tonAirBeforeStart2(IN:=eRunningStateFeeder=E_WickFeederSorterState.eSorting, PT:=T#2S);
tonAirAfterStop(IN:=eRunningStateFeeder=E_WickFeederSorterState.eSleeveFull, PT:=T#2S);

tonbSeparatorPos1AndNotbWickAtSleve1(IN:=bSeparatorPos1 AND NOT bWickAtSleve1,PT:=T#3S);
tonbSeparatorPos2AndNotbWickAtSleve2(IN:=bSeparatorPos2 AND NOT bWickAtSleve2,PT:=T#3S);
tonbSeparatorPos1(IN:=bSeparatorPos1,PT:=T#300MS);
tonbSeparatorPos2(IN:=bSeparatorPos2,PT:=T#300MS);

tobbSleve1SeparatorIn(IN:=bSleve1SeparatorIn,PT:=T#1S);
tobbSleve2SeparatorIn(IN:=bSleve2SeparatorIn,PT:=T#1S);
fbbQueFullAtSleve1 (bIN:=	bQueFullAtSleve1,	tFilterTimeOn:=T#300MS, tFilterTimeOff:=T#300MS, 	bOUT=> );										
fbbQueFullAtSleve2 (bIN:=	bQueFullAtSleve2,	tFilterTimeOn:=T#300MS, tFilterTimeOff:=T#300MS, 	bOUT=> );										
fbbWickAtPipe 		(bIN:=	bWickAtPipe,		tFilterTimeOn:=T#100MS, tFilterTimeOff:=T#30MS,		bOUT=> );	
fbbNotWickAtPipe 	(bIN:=	NOT bWickAtPipe AND iSortingCase=35,		tFilterTimeOn:=T#2S, tFilterTimeOff:=T#100MS,		bOUT=> );	
									
tonCaseA			(IN:=iSortingCase = 20 , PT:=T#600MS);
tonCaseB			(IN:=iSortingCase = 35 , PT:=T#300MS);
tonCaseC			(IN:=iSortingCase = 20 , PT:=T#600MS);
tonCaseD			(IN:=iSortingCase = 20 , PT:=T#600MS);
//prszesunęcie wartosci czujnika po buforu opoznenia 

TimerOn (IN := NOT bImpOn, PT := T#10MS);
IF TimerOn.Q THEN
	bImpOn := TRUE;
END_IF
TimerOff (IN := bImpOn, PT := T#10MS);
IF TimerOff.Q THEN
	bImpON := FALSE;
END_IF

tonHammer1Down(IN:= bHammer1Down, PT:=T#200MS);
tonHammer2Down(IN:= bHammer2Down, PT:=T#200MS);

(** Dodatkowy timer przy zatrzymywaniu**)
tonStoppingTime( IN:= eState= E_Station.eStopping, PT:=T#2S);
END_ACTION

ACTION ACT_Warning:
 //Warning czujnik poziomu	
 	tonLowLevelSensor( IN:=( NOT  bWheelLevelSensor (*OR NOT bQueFullAfterWheelSensor*) OR NOT bQueFullSensor) AND bRun, PT:= T#5S);
 	
 	IF tonLowLevelSensor.Q THEN
 		bWarning				:= TRUE;
	ELSE
		bWarning				:= FALSE;
 	END_IF
END_ACTION

END_FUNCTION_BLOCK

// ---- POUs/P08_CapSorter.TcPOU
(*
Nazwa:			P08_CapFeeder
Opis:			Stacja podajnika nasadek
Wersja:			v0.2
Data:			2024-01-12
Autor:			DP
Urzadzenia:		
Konfiguracja:	
Info:

*)
PROGRAM P08_CapSorter
VAR_INPUT
	IbCapSorterGateScrewerSensor 			:BOOL;			
	IbCapSorterGateWeightSensor				:BOOL;
	//WEJSCIA I WYJSCIA SPRZETOWE
	IbCapSorterDragHomingSensor 			 :BOOL;						// Czujnik bazowania
	QbCapSorterDragActuator               	 :BOOL;						// Siłownikiem przeciągania 
	IbCapSorterDragUpSensor 				 :BOOL;						// Czujnik
	IbCapSorterDragDownSensor 				 :BOOL;						// Czujnik
	                                         
	QbCapSorterDragLeadBefore1Actuator       :BOOL;						// Siłownikiem prowadzenia przed 
	IbCapSorterDragLeadBefore1UpSensor 	 	 :BOOL;						// Czujnik
 	IbCapSorterDragLeadBefore2UpSensor 	 	 :BOOL;						// Czujnik			
	QbCapSorterDragLeadAfter1Actuator        :BOOL;						// Siłownikiem prowadzenia za
	IbCapSorterDragLeadAfter1UpSensor 	 	 :BOOL;						// Czujnik
 	IbCapSorterDragLeadAfter2UpSensor 	 	 :BOOL;						// Czujnik			

END_VAR
VAR
	
	(*******PRZECIAGANIE**********)
	eCapSorterDragStation						: E_Station;
	eCapSorterDragRunningStation				: E_DragStationState;
	fbCapSorterDragState						: FB_State;
	fbCapSorterDragStation						: FB_FormsDragStepper;	
	
	

	
	
	//Pomocnicze
	tofCapSorterDragEnable					: TOF;
	
	//Stoper
	QbCapSorterStoperActuator				: BOOL;				// bit to wysterowania sygnału stopera	
	tpStoperTimerOn							: TP;				// timer do generowania impulsu
	fbStoperSensorDelay						: FB_InputFilter;	// filtr do generowania sygnału 
	lrCapSorterStoperPosition						: LREAL;	
	rtCapSorterStoperDraging: R_TRIG;
	rtCapSorterStoperEndingOfDraging: R_TRIG;	
	//Inne
	bTemp: BOOL;

	rtCapSorterStoperPackMLStarting: R_TRIG;
	bCapSorterStoperWaitingForSensor: BOOL;
	bCapSorterStoperActuatorDelay: BOOL;
	tonbCapSorterStoperActuatorDelay: TON;
	
	//ManualStoper
	rtManualMode	: R_TRIG;
	ftManualMode	: F_TRIG;	
	bCapSorterStoperActuatorLastState	:BOOL;
	
END_VAR

//bCapSorterDisable:=VIS.bCapPuttedCheckIgnoreErrors;


tofCapSorterDragEnable(IN:= GVL.bCapSorterDragEnable, PT:= T#5S);
aLimits();
aStoper();
aDragStation();
aCapSorterWarnings();


(********* GENEROWANIE STANU STACJI DO WIZKI**********)
fbCapSorterDragState(
	eState:=eCapSorterDragStation, 
	bRun:=VIS.bCapSorterDragRun,
	eFormsDragingRunningState:=eCapSorterDragRunningStation, 
	sStateDesc=> VIS.sCapSorterDragState,
	iState=>VIS.iCapSorterDragState);
(***** KONIEC GENEROWANIE STANU STACJI DO WIZKI*******)



IF fbCapSorterDragStation.bCycleDone AND bManualMode THEN
	VIS.bCapSorterDragRun 						:= FALSE;
	GVL.bCapSorterDragPrepareRun				:= FALSE;
END_IF

ACTION aCapSorterWarnings:

//Warning 0
IF stCapSorterRead.eReservedSignals.iReserved20.0 AND NOT CapSorterWarning[0].bWarning THEN
	CapSorterWarning[0].bWarning										:=TRUE;
	CapSorterWarning[0].udiWarningCode									:=41;
	CapSorterWarning[0].sDescription									:='Sorter nasadek | Brak nasadek w zasobniku';
ELSIF NOT stCapSorterRead.eReservedSignals.iReserved20.0 THEN//AND CapSorterWarning[0].bAcknowledge THEN
	CapSorterWarning[0].bWarning										:=FALSE;
	CapSorterWarning[0].bAcknowledge									:=FALSE;
	VIS.uliWarningAcknowledge.27										:=FALSE;
ELSIF CapSorterWarning[0].bAcknowledge THEN                               
	CapSorterWarning[0].bAcknowledge									:=TRUE;
END_IF

//Warning 1
IF stCapSorterRead.eReservedSignals.iReserved20.1 AND NOT CapSorterWarning[1].bWarning THEN
	CapSorterWarning[1].bWarning										:=TRUE;
	CapSorterWarning[1].udiWarningCode									:=42;
	CapSorterWarning[1].sDescription									:='Sorter nasadek | Brak nasadek na stole - sprawdź transporter pośredni';
ELSIF NOT stCapSorterRead.eReservedSignals.iReserved20.1 AND CapSorterWarning[1].bAcknowledge THEN
	CapSorterWarning[1].bWarning										:=FALSE;
	CapSorterWarning[1].bAcknowledge									:=FALSE;
	VIS.uliWarningAcknowledge.28										:=FALSE;
ELSIF CapSorterWarning[1].bAcknowledge THEN
	CapSorterWarning[1].bAcknowledge									:=TRUE;
END_IF

//Warning 2
IF stCapSorterRead.eReservedSignals.iReserved20.2 AND NOT CapSorterWarning[2].bWarning THEN
	CapSorterWarning[2].bWarning										:=TRUE;
	CapSorterWarning[2].udiWarningCode									:=43;
	CapSorterWarning[2].sDescription									:='Sorter nasadek | Niepobrana nasadka przez chwytak 1';
ELSIF NOT stCapSorterRead.eReservedSignals.iReserved20.1 AND CapSorterWarning[2].bAcknowledge THEN
	CapSorterWarning[2].bWarning										:=FALSE;
	CapSorterWarning[2].bAcknowledge									:=FALSE;
	VIS.uliWarningAcknowledge.29										:=FALSE;
ELSIF CapSorterWarning[2].bAcknowledge THEN
	CapSorterWarning[2].bAcknowledge									:=TRUE;
END_IF

//Warning 3
IF stCapSorterRead.eReservedSignals.iReserved20.3 AND NOT CapSorterWarning[3].bWarning THEN
	CapSorterWarning[3].bWarning										:=TRUE;
	CapSorterWarning[3].udiWarningCode									:=44;
	CapSorterWarning[3].sDescription									:='Sorter nasadek | Niepobrana nasadka przez chwytak 2';
ELSIF NOT stCapSorterRead.eReservedSignals.iReserved20.1 AND CapSorterWarning[3].bAcknowledge THEN
	CapSorterWarning[3].bWarning										:=FALSE;
	CapSorterWarning[3].bAcknowledge									:=FALSE;
	VIS.uliWarningAcknowledge.30										:=FALSE;
ELSIF CapSorterWarning[3].bAcknowledge THEN
	CapSorterWarning[3].bAcknowledge									:=TRUE;
END_IF

//Warning 4
IF stCapSorterRead.eReservedSignals.iReserved20.4 AND NOT CapSorterWarning[4].bWarning THEN
	CapSorterWarning[4].bWarning										:=TRUE;
	CapSorterWarning[4].udiWarningCode									:=45;
	CapSorterWarning[4].sDescription									:='Sorter nasadek | Niepobrana nasadka przez chwytak 3';
ELSIF NOT stCapSorterRead.eReservedSignals.iReserved20.1 AND CapSorterWarning[4].bAcknowledge THEN
	CapSorterWarning[4].bWarning										:=FALSE;
	CapSorterWarning[4].bAcknowledge									:=FALSE;
	VIS.uliWarningAcknowledge.31										:=FALSE;
ELSIF CapSorterWarning[4].bAcknowledge THEN
	CapSorterWarning[4].bAcknowledge									:=TRUE;
END_IF

//Warning 5
IF stCapSorterRead.eReservedSignals.iReserved20.5 AND NOT CapSorterWarning[5].bWarning THEN
	CapSorterWarning[5].bWarning										:=TRUE;
	CapSorterWarning[5].udiWarningCode									:=46;
	CapSorterWarning[5].sDescription									:='Sorter nasadek | Niepobrana nasadka przez chwytak 4';	
ELSIF NOT stCapSorterRead.eReservedSignals.iReserved20.1 AND CapSorterWarning[5].bAcknowledge THEN
	CapSorterWarning[5].bWarning										:=FALSE;
	CapSorterWarning[5].bAcknowledge									:=FALSE;
	VIS.uliWarningAcknowledge.32										:=FALSE;
ELSIF CapSorterWarning[5].bAcknowledge THEN
	CapSorterWarning[5].bAcknowledge									:=TRUE;
END_IF
END_ACTION

ACTION aDragStation:
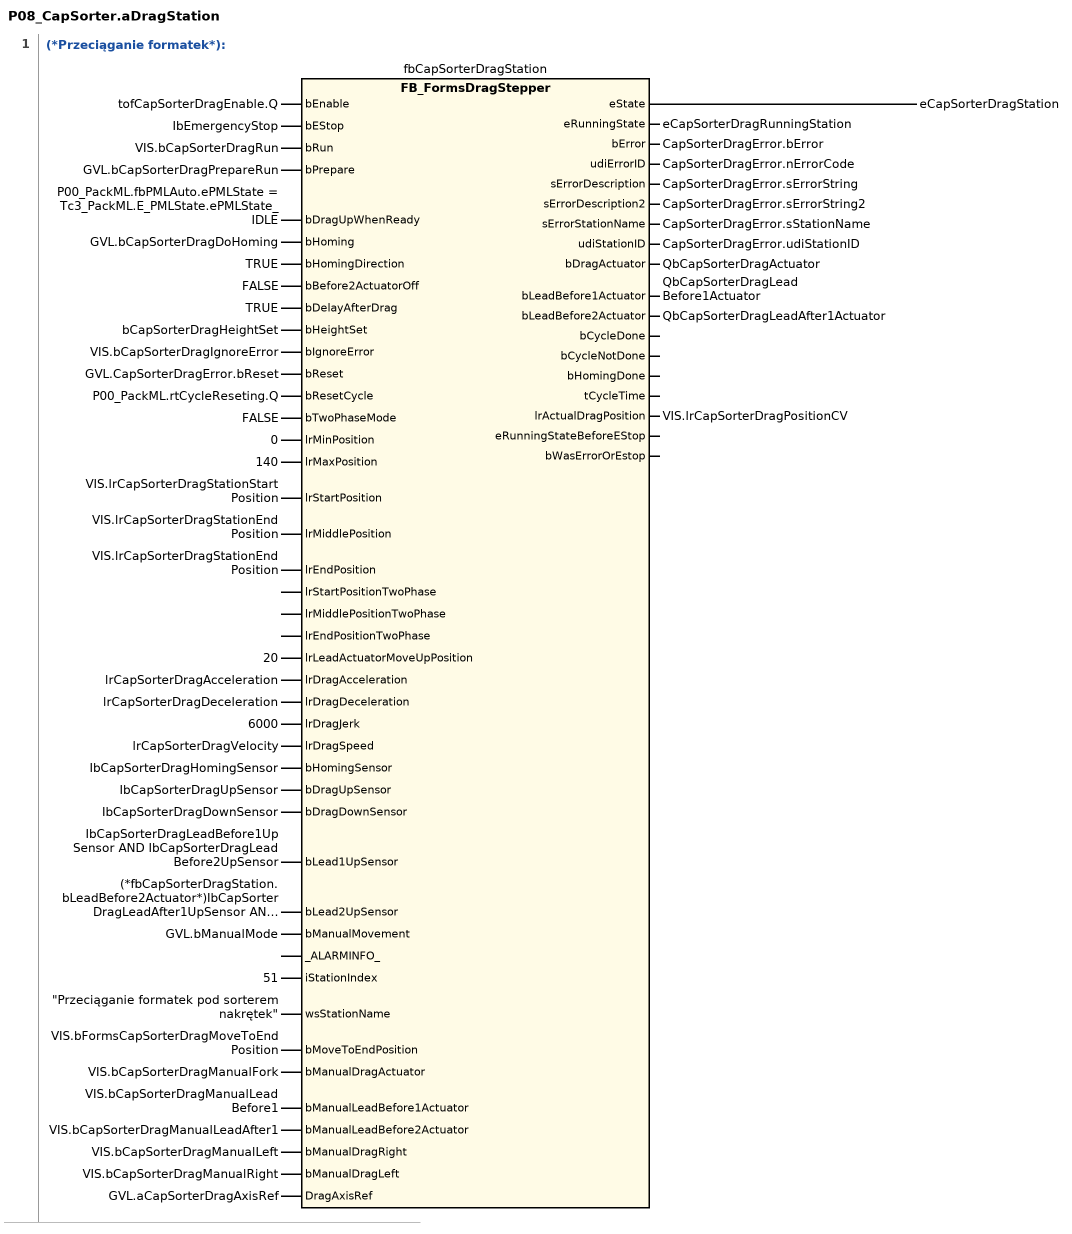
// NETWORK 1
// label: (*Przeciąganie formatek*)
fbCapSorterDragStation(
    bEnable := tofCapSorterDragEnable.Q,
    bEStop := IbEmergencyStop,
    bRun := VIS.bCapSorterDragRun,
    bPrepare := GVL.bCapSorterDragPrepareRun,
    bDragUpWhenReady := P00_PackML.fbPMLAuto.ePMLState = Tc3_PackML.E_PMLState.ePMLState_IDLE,
    bHoming := GVL.bCapSorterDragDoHoming,
    bHomingDirection := TRUE,
    bBefore2ActuatorOff := FALSE,
    bDelayAfterDrag := TRUE,
    bHeightSet := bCapSorterDragHeightSet,
    bIgnoreError := VIS.bCapSorterDragIgnoreError,
    bReset := GVL.CapSorterDragError.bReset,
    bResetCycle := P00_PackML.rtCycleReseting.Q,
    bTwoPhaseMode := FALSE,
    lrMinPosition := 0,
    lrMaxPosition := 140,
    lrStartPosition := VIS.lrCapSorterDragStationStartPosition,
    lrMiddlePosition := VIS.lrCapSorterDragStationEndPosition,
    lrEndPosition := VIS.lrCapSorterDragStationEndPosition,
    lrLeadActuatorMoveUpPosition := 20,
    lrDragAcceleration := lrCapSorterDragAcceleration,
    lrDragDeceleration := lrCapSorterDragDeceleration,
    lrDragJerk := 6000,
    lrDragSpeed := lrCapSorterDragVelocity,
    bHomingSensor := IbCapSorterDragHomingSensor,
    bDragUpSensor := IbCapSorterDragUpSensor,
    bDragDownSensor := IbCapSorterDragDownSensor,
    bLead1UpSensor := IbCapSorterDragLeadBefore1UpSensor AND IbCapSorterDragLeadBefore2UpSensor,
    bLead2UpSensor := (*fbCapSorterDragStation.bLeadBefore2Actuator*)IbCapSorterDragLeadAfter1UpSensor AND IbCapSorterDragLeadAfter2UpSensor,
    bManualMovement := GVL.bManualMode,
    iStationIndex := 51,
    wsStationName := "Przeciąganie formatek pod sorterem nakrętek",
    bMoveToEndPosition := VIS.bFormsCapSorterDragMoveToEndPosition,
    bManualDragActuator := VIS.bCapSorterDragManualFork,
    bManualLeadBefore1Actuator := VIS.bCapSorterDragManualLeadBefore1,
    bManualLeadBefore2Actuator := VIS.bCapSorterDragManualLeadAfter1,
    bManualDragRight := VIS.bCapSorterDragManualLeft,
    bManualDragLeft := VIS.bCapSorterDragManualRight,
    DragAxisRef := GVL.aCapSorterDragAxisRef,
    eRunningState => eCapSorterDragRunningStation,
    bError => CapSorterDragError.bError,
    udiErrorID => CapSorterDragError.nErrorCode,
    sErrorDescription => CapSorterDragError.sErrorString,
    sErrorDescription2 => CapSorterDragError.sErrorString2,
    sErrorStationName => CapSorterDragError.sStationName,
    udiStationID => CapSorterDragError.udiStationID,
    bDragActuator => QbCapSorterDragActuator,
    bLeadBefore1Actuator => QbCapSorterDragLeadBefore1Actuator,
    bLeadBefore2Actuator => QbCapSorterDragLeadAfter1Actuator,
    lrActualDragPosition => VIS.lrCapSorterDragPositionCV); // FB_FormsDragStepper
eCapSorterDragStation := fbCapSorterDragStation.eState;
END_ACTION

ACTION aLimits:
//
IF 	VIS.lrCapSorterDragStationStartPosition		= 0		THEN	VIS.lrCapSorterDragStationStartPosition	:=	7;		END_IF;
IF 	VIS.lrCapSorterDragStationEndPosition		= 0		THEN	VIS.lrCapSorterDragStationEndPosition		:=	142;	END_IF;
END_ACTION

ACTION aStoper:
(*
Nazwa:			aStoper
Opis:			Stoper spowalniania formatek
Wersja:			v0.1
Data:			2024-03-21
Autor:			DP
Urzadzenia:		
Konfiguracja:	
Info:

*)


// 0 - Przliczanie od predkości przeciagania				   
lrCapSorterStoperPosition	 :=	(188.25 * EXPT(lrCapSorterDragVelocity,-0.404));
	

// 1 - Wysuwanie stopera na koniec przesuwania gdy pracuje
rtCapSorterStoperDraging(CLK:=  
								P08_CapSorter.fbCapSorterDragStation.eRunningState = E_DragStationState.eDraging AND 
								((P00_PackML.fbPMLAuto.ePMLState = E_PMLState.ePMLState_STOPPING) OR  (P00_PackML.fbPMLAuto.ePMLState = E_PMLState.ePMLState_EXECUTE)) AND
						   		P08_CapSorter.fbCapSorterDragStation.lrActualDragPosition > lrCapSorterStoperPosition+20 
						,Q=>);
						
IF rtCapSorterStoperDraging.Q THEN
	QbCapSorterStoperActuator	:= TRUE;
END_IF


									
// 2 - Sygnał czekania na czujnik formatek
rtCapSorterStoperPackMLStarting (CLK:=  	
											(P00_PackML.fbPMLAuto.ePMLState = E_PMLState.ePMLState_STARTING)
								,Q=>);

								

//rtCapSorterStoperEndingOfDraging(CLK:=  	P08_CapSorter.fbCapSorterDragStation.eRunningState = E_DragStationState.eDraged AND 
rtCapSorterStoperEndingOfDraging(CLK:=  	P08_CapSorter.fbCapSorterDragStation.eRunningState = E_DragStationState.eDragingDone AND 
											((P00_PackML.fbPMLAuto.ePMLState = E_PMLState.ePMLState_STOPPING) OR  (P00_PackML.fbPMLAuto.ePMLState = E_PMLState.ePMLState_EXECUTE))
								,Q=>);
						

IF rtCapSorterStoperEndingOfDraging.Q OR rtCapSorterStoperPackMLStarting.Q THEN
	bCapSorterStoperWaitingForSensor	:=	TRUE;	
END_IF							

// 3 - Wyłączanie stopera
IF NOT bDosingTwoPhases THEN
	IF bCapSorterStoperWaitingForSensor AND P00_PackML.fbIbCapSorterFourthFormCheckFormSensor.bOut THEN	
		bCapSorterStoperActuatorDelay	:=	TRUE;
	END_IF
ELSE
	IF bCapSorterStoperWaitingForSensor (*AND MAIN.IbCapSorterFourthFormCheckFormSensor*) AND iCapSorterDragFormCounter >=1 AND P00_ReadRFIDCard.bReadedCardCapSorter THEN	
		bCapSorterStoperActuatorDelay	:=	TRUE;
	END_IF
END_IF

IF 	nFormTransportersBeforeScrewerVelocitySV < 610 AND NOT bDosingTwoPhases THEN
	tonbCapSorterStoperActuatorDelay(IN:=bCapSorterStoperActuatorDelay, PT:=T#1S150MS);
ELSE
	tonbCapSorterStoperActuatorDelay(IN:=bCapSorterStoperActuatorDelay, PT:=T#790MS);//990
END_IF

IF tonbCapSorterStoperActuatorDelay.Q THEN
	bCapSorterStoperActuatorDelay		:=	FALSE;
	bCapSorterStoperWaitingForSensor	:=	FALSE;
	QbCapSorterStoperActuator			:=	FALSE;
END_IF


//Manual
rtManualMode	(CLK:=bManualMode,	Q=>);
ftManualMode	(CLK:=bManualMode,	Q=>);
IF rtManualMode.Q THEN
	bCapSorterStoperActuatorLastState	:=	QbCapSorterStoperActuator;
	VIS.bCapSorterStoperManualActuator	:=	QbCapSorterStoperActuator;
END_IF
IF bManualMode THEN
	QbCapSorterStoperActuator			:=	VIS.bCapSorterStoperManualActuator;
END_IF
IF ftManualMode.Q THEN
	QbCapSorterStoperActuator			:= bCapSorterStoperActuatorLastState;
END_IF
// Koniec Manual
END_ACTION

END_PROGRAM

// ---- POUs/P01_PucksInserter.TcPOU
(*
Nazwa:			P01_PucksInserter
Opis:			Stacja podajnika opakowań
Wersja:			v0.1
Data:			2025-02-04
Autor:			DP
Urzadzenia:		
Konfiguracja:	
Info:

*)
PROGRAM P01_PucksInserter
VAR_INPUT

	//52N6.1 Pneumatyka IO
	IbPucksInserterLevelSensor					:BOOL;			// Czujnik kolejki butelki
	IbPucksInserterWheelEntrySensor				:BOOL;			// Czujnik   pierwszego slotu w karuzeli (to 
	IbPucksInserterWheelExitSensor				:BOOL;			// Czujnik
	IbPucksInserterFormGateBeforeSensor 		:BOOL;			// Czujnik przed szlabanem formatek
	IbPucksInserterFormGateAfterSensor 			:BOOL;			// Czujnik za szlabanem formatek	
 	IbPucksInserterHammerUpSensor				:BOOL;			// Czujnik położenia siłownika - góra
	IbPucksInserterHammerDownSensor				:BOOL;			// Czujnik polożenia siłowniak - dół
	IbPucksInserterTrayOnSensor					:BOOL;			// Czujnik tacka wysunieta
	//52N6.2 Pneumatyka IO	
	IbPucksInserterTrayOffSensor				:BOOL;			// Czujnik tacka schowana
	IbPucksInserterFormPositioningOnSensor		:BOOL;			// Czujnik wysuniecia siłownika pozycjonujacego formatke
	IbPucksInserterFormPositioningOffSensor		:BOOL;			// Czujnik schowania siłownika pozycjonujacego formatke
	IbPucksInserterGate1OnSensor				:BOOL;			// Czujnik otwarcia 1 szlabanu (Lewy)
	IbPucksInserterGate1OffSensor				:BOOL;			// Czujnik zamknięcia 1 szlabanu (Lewy) 
	IbPucksInserterGate2OnSensor				:BOOL;			// Czujnik otwarcia 2 szlabanu 
	IbPucksInserterGate2OffSensor				:BOOL;			// Czujnik zamknięcia 2 szlabanu (Prawy) 
	IbPucksInserterHomingSensor					:BOOL;			// Czujnik bazowania
	
	//Inne
	IbPucksInserterNotInsertedSensor			:BOOL;			// Czujnik źle włozonej butelki za stacją	
	
	IbPucksInserterPushTablesSensor				:BOOL;
END_VAR

VAR

	//BC3 
	IbPucksInserterFuseDrivesOK					AT %I*: BOOL; 			// Zabezpieczenie serwa
	IbPucksInserterTransporter1OK				AT %I*: BOOL; 			// Bezpiecznik silnikowe napędu transportera 1
	IbPucksInserterTransporter2OK				AT %I*: BOOL; 			// Bezpiecznik silnikowe napędu transportera 2	
	IbPucksInserterFuseFB1OK					AT %I*: BOOL;			// Bezpiecznik FB1 przepalony
	QbPucksInserterHammerHeightUpCmd 			AT %Q*: BOOL; 			// Wyjście sterujące podnośnikiem
	QbPucksInserterHammerHeightDownCmd 			AT %Q*: BOOL; 			// Wyjście sterujące podnośnikiem
	//GVL_IO QbPickInserterDoorsClose			AT %Q*:BOOL;			// Rozkaz zamkniecia
	QudiPucksInserterHammerHeightEncoderSetCV	AT %Q*: UDINT;			// Enkoder - Set Counter value
	QbPucksInserterHammerHeightEncoderSetC		AT %Q*: BOOL; 			// Enkoder - Set Counter 
	IudiPucksInserterHammerHeightEncoderCV 		AT %I*: UDINT;	 		// Enkoder - Counter value
	IbPucksInserterHammerHeightEncoderSetCDone	AT %I*: BOOL; 			// Enkoder - Set Counter done

	//DI5
	//GVL_IO IbPucksInserterDoorsOpen	{warning 'PI'}	AT %I*	:BOOL;	//Otwarte drzwi podajnika opakowań
	//GLV_IO etop 0
	//GLV_IO etop 1
	//GLV_IO stop
	//GLV_IO start
	//Safety reset

	//DO4
	//Lamps green
	//Lamps blue

	fbPucksInserter						  	: FB_PucksInserter;		// Bloczek do obsługi stacji podajnika butelek
	fbTurnTable								: FB_MitsubishiInverter; 	//Bloczek do obsługi falownika stołu obrotewego
	
	ePucksInserterStationState				: E_Station;
	ePucksInserterRunningState				: E_PuckInserterState;
	fbPucksInserterState					: FB_State;
	
	ePucksInserterTurnTableState			: E_Station;
	ePucksInserterTurnTableRunningState		: E_ConveyorState;
	fbBottleSorterTurnTableState			: FB_State;
	
	fbGatePucksInserter						: FB_SpringGateV2;
	
	//Wyjścia sterujące
	QbPucksInserterHammer					:BOOL;			// Wbijak
	QbPucksInserterTray						:BOOL;			// Ruchomy blat (tacka)
	QbPucksInserterGate1					:BOOL;			// Szlaban 1 (lewy)
	QbPucksInserterGate2					:BOOL;			// Szlaban 2 (prawy)
	QbPucksInserterFormGate					:BOOL;			// Szlaban formatki
	QbPucksInserterFormPositioning			:BOOL;			// Pozycjonowanie formatki

	// Stół obrotowy
	uiPucksInserterTurnTableSW					AT %I*: UINT;
	uiPucksInserterTurnTableActualVelocity		AT %I*: UDINT;
	uiPucksInserterTurnTableCW  				AT %Q*: UINT;
	udiPucksInserterTurnTableVelocity			AT %Q*: UDINT;
	
	// Transporter
	uiPucksInserterConveyorSW					AT %I*: UINT;
	uiPucksInserterConveyorActualVelocity		AT %I*: UDINT;
	uiPucksInserterConveyorCW  					AT %Q*: UINT;
	udiPucksInserterConveyorVelocity			AT %Q*: UDINT;	
	IbPucksInserterConveyorWcState				AT %I*: BOOL;
	
	// Serwo
	// GVL axis
	diPucksInserterWheelZPhaseOffset			AT %I*: DINT; // Offset serwa Z


	// Bazowanie
	tonPucksInserterEnable	: TON;
	rtEnable	: R_TRIG;
	
	//testowe
	bTest :BOOL;
	bTest2 :BOOL;	
	bTestHomingPI:BOOL;
	bPITest:BOOL;
	 
	//Stół pchający    //Vasyl 27.05
	fbPushTable_m1: FB_MitsubishiInverter;
	fbPushTable_m2: FB_MitsubishiInverter;
	fbPushTable_m3: FB_MitsubishiInverter;	
	
	QnPucksInserterPushTable_m1_VelocitySV 						AT %Q*: UDINT; 	
	InPucksInserterPushTable_m1_VelocityCV 						AT %I*: UDINT;	
	InPucksInserterPushTable_m1_STW 							AT %I*: UINT; 	
	QnPucksInserterPushTable_m1_CTW 							AT %Q*: UINT;  	
	InPucksInserterPushTable_m1_ErrorCode 						AT %I*: UINT;	
	
	QnPucksInserterPushTable_m2_VelocitySV 						AT %Q*: UDINT; 	
	InPucksInserterPushTable_m2_VelocityCV 						AT %I*: UDINT;	
	InPucksInserterPushTable_m2_STW 							AT %I*: UINT; 
	QnPucksInserterPushTable_m2_CTW 							AT %Q*: UINT;  	
	InPucksInserterPushTable_m2_ErrorCode 						AT %I*: UINT;	
	
	QnPucksInserterPushTable_m3_VelocitySV 						AT %Q*: UDINT; 	
	InPucksInserterPushTable_m3_VelocityCV 						AT %I*: UDINT; 	
	InPucksInserterPushTable_m3_STW 							AT %I*: UINT; 
	QnPucksInserterPushTable_m3_CTW 							AT %Q*: UINT;  	
	InPucksInserterPushTable_m3_ErrorCode 						AT %I*: UINT;	

	
	fbPucksInserterPushTableState			: FB_State;
	ePucksInserterPushTableState			: E_Station;
	ePucksInserterPushTableRunningState		: E_PuckInserterState;
	
	fbPucksInserterPushTableRollerState			: FB_State;
	ePucksInserterPushTableRollerState			: E_Station;
	ePucksInserterPushTableRollerRunningState	: E_PuckInserterState;
END_VAR

aWarning();
aPucksInserter();
aTurntable(); 
aGateTime();
aGate();
aPushTable();

//VIS.nPucksInserterTurnTableVelocityCV := uiPucksInserterTurnTableActualVelocity;
VIS.nPucksInserterConveyorVelocityCV:=uiPucksInserterConveyorActualVelocity;
VIS.uiPucksInserterPushTable_m1_Velocity:=UDINT_TO_INT(InPucksInserterPushTable_m1_VelocityCV);
VIS.uiPucksInserterPushTable_m2_Velocity:=UDINT_TO_INT(InPucksInserterPushTable_m2_VelocityCV);
VIS.uiPucksInserterPushTable_m3_Velocity:=UDINT_TO_INT(InPucksInserterPushTable_m3_VelocityCV);

(* BAZOWANIE - ZMIAN*)
tonPucksInserterEnable (IN:=fbPucksInserter.bEnable,PT:=T#5S); (*Dodany ton bo Wizka zjebnie wgrywa zmienne, najpierw włacza Enabla a potem dopiero wybiera recepture*)
rtEnable(CLK:=tonPucksInserterEnable.Q,Q=>);
IF rtEnable.Q AND (P00_PackML.fbPMLAuto.ePMLState = E_PMLState.ePMLState_IDLE OR P00_PackML.fbPMLAuto.ePMLState = E_PMLState.ePMLState_EXECUTE)   THEN
	VIS.bPucksInserterHeightSet:=TRUE;
ELSIF fbPucksInserter.eState=E_Station.eHomingDone  OR VIS.bErrorOccure THEN
 	VIS.bPucksInserterHeightSet:=FALSE;
END_IF
(*KONIEC BAZOWANIE - ZMIANA*)


(********KASOWANIE ROZKAZÓW CYKLI*********)
IF fbPucksInserter.bCycleDone AND bManualMode THEN
	VIS.bPucksInserterRun := FALSE;
END_IF

(*
IF bPITest AND NOT VIS.bPucksInserterRun THEN
	VIS.bPucksInserterRun := TRUE;
END_IF
IF VIS.bPucksInserterRun AND bPITest AND fbPucksInserter.bCycleDone THEN
	VIS.bPucksInserterRun := FALSE;	
END_IF*)


fbPucksInserterState(
	eState									:= ePucksInserterStationState,
	bRun									:= VIS.bPucksInserterRun,
	eBottleSorterRunningState				:= ePucksInserterRunningState,
	sStateDesc								=> VIS.sPucksInserterState,
	iState									=> VIS.iPucksInserterState);
	
fbPucksInserterPushtableState(
	eState									:= ePucksInserterPushTableState,
    bRun						            := gvl.bPucksInserterPushTable_m1_Run OR vis.bPucksInserterPushTable_m1_ManualCmdStart,
    eBottleSorterRunningState	            := ePucksInserterPushTableRunningState,
    sStateDesc					            => VIS.sPucksInserterPushTableState,
    iState						            => VIS.iPucksInserterPushTableState);
	
fbPucksInserterPushTableRollerState(
	eState									:= ePucksInserterPushTableRollerState,	
    bRun						            := gvl.bPucksInserterPushTable_m2_Run OR vis.bPucksInserterPushTable_m2_ManualCmdStart,	
    eBottleSorterRunningState	            := ePucksInserterPushTableRollerRunningState,	
    sStateDesc					            => VIS.sPucksInserterPushTableRollerState,	
    iState						            => VIS.iPucksInserterPushTableRollerState);

ACTION aGate:
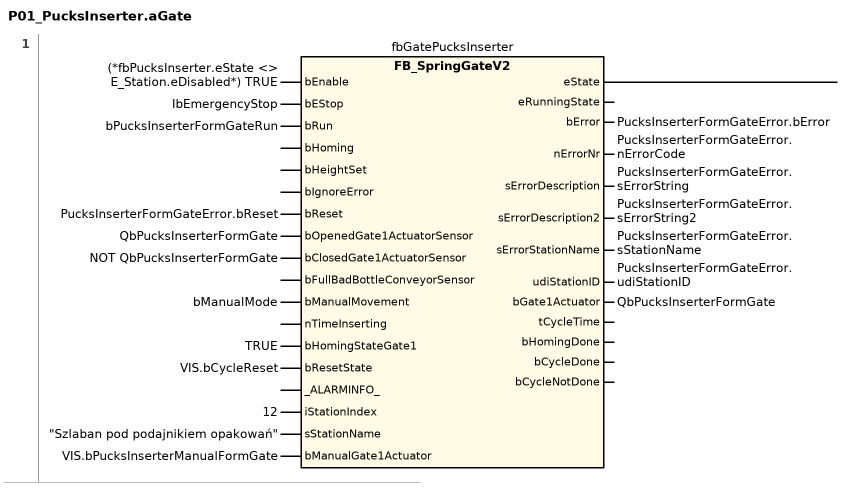
// NETWORK 1
fbGatePucksInserter(
    bEnable := (*fbPucksInserter.eState <> E_Station.eDisabled*) TRUE,
    bEStop := IbEmergencyStop,
    bRun := bPucksInserterFormGateRun,
    bReset := PucksInserterFormGateError.bReset,
    bOpenedGate1ActuatorSensor := QbPucksInserterFormGate,
    bClosedGate1ActuatorSensor := NOT QbPucksInserterFormGate,
    bManualMovement := bManualMode,
    bHomingStateGate1 := TRUE,
    bResetState := VIS.bCycleReset,
    iStationIndex := 12,
    sStationName := "Szlaban pod podajnikiem opakowań",
    bManualGate1Actuator := VIS.bPucksInserterManualFormGate,
    bError => PucksInserterFormGateError.bError,
    nErrorNr => PucksInserterFormGateError.nErrorCode,
    sErrorDescription => PucksInserterFormGateError.sErrorString,
    sErrorDescription2 => PucksInserterFormGateError.sErrorString2,
    sErrorStationName => PucksInserterFormGateError.sStationName,
    udiStationID => PucksInserterFormGateError.udiStationID,
    bGate1Actuator => QbPucksInserterFormGate); // FB_SpringGateV2
END_ACTION

ACTION aGateTime:
IF bFormTransportersDispencerSlowSpeed THEN 
	fbGatePucksInserter.nTimeInserting	:=	350; //500 pomieszane zwalnianie transportera??
ELSE
	fbGatePucksInserter.nTimeInserting	:=	350;	//400
END_IF
END_ACTION

ACTION aPucksInserter:
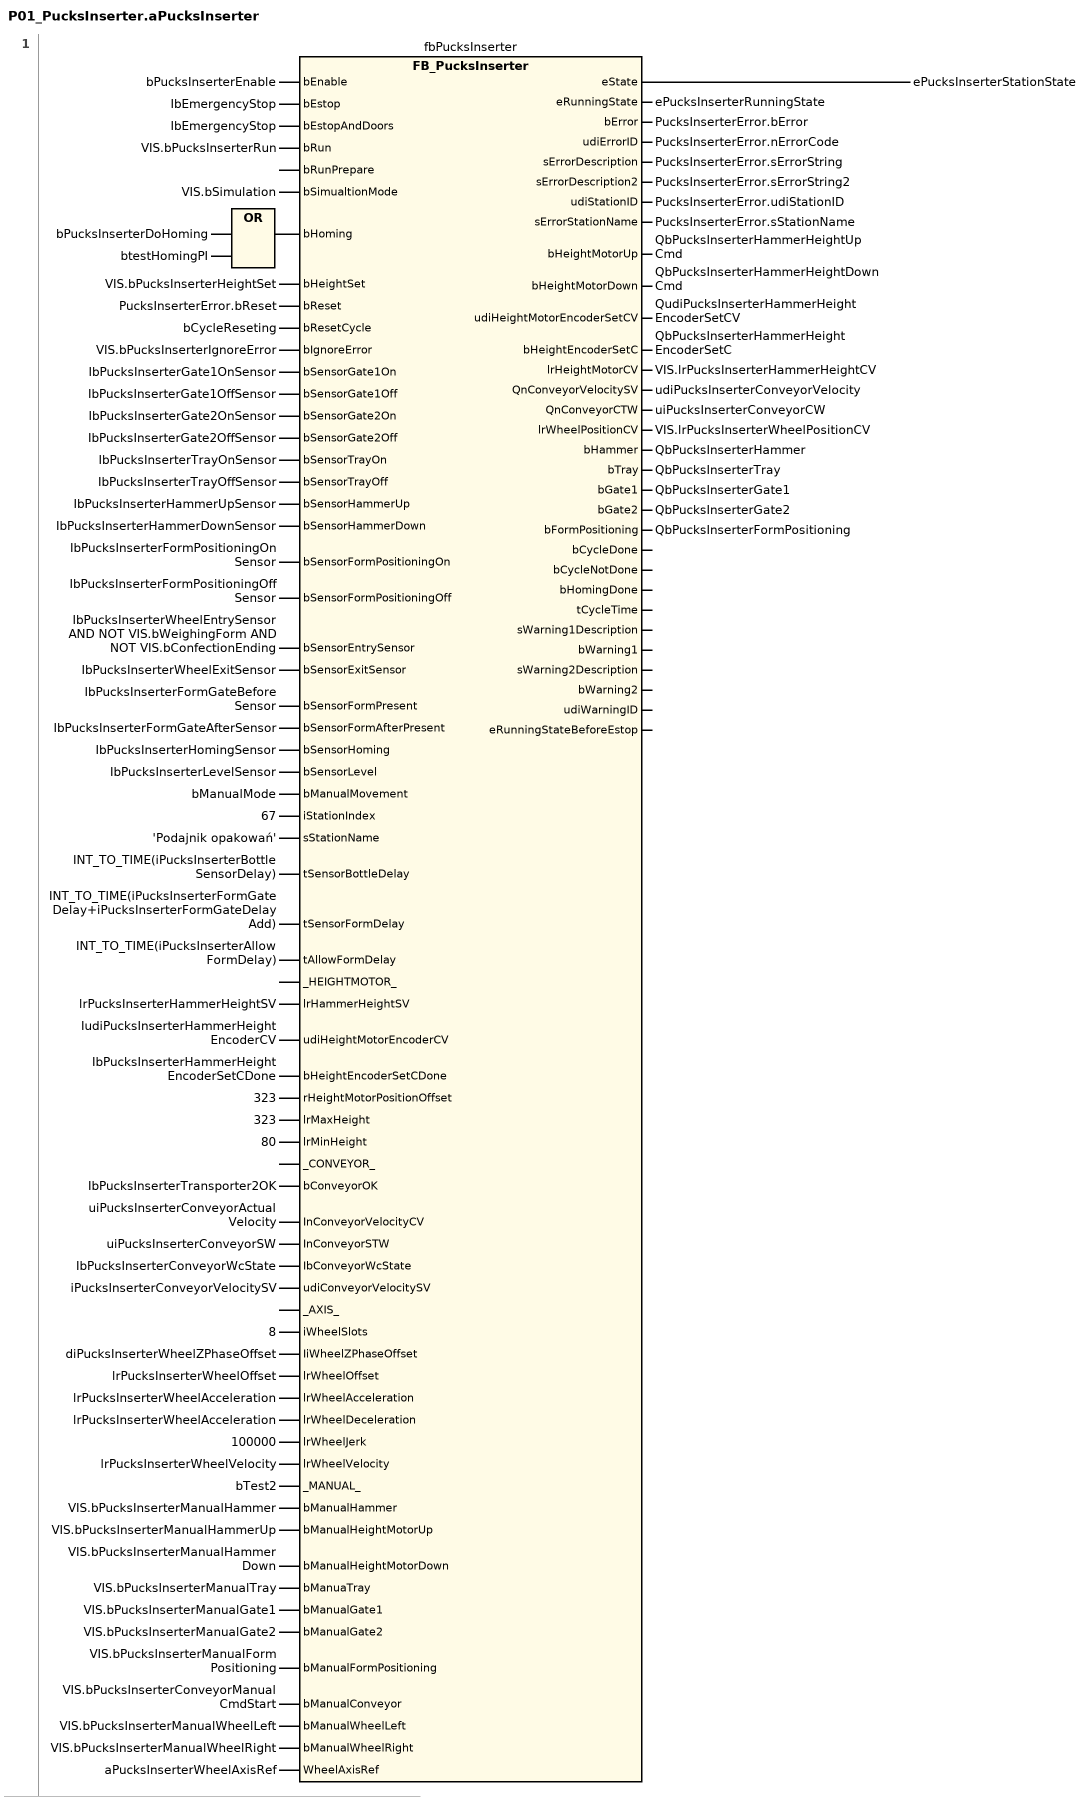
// NETWORK 1
fbPucksInserter(
    bEnable := bPucksInserterEnable,
    bEstop := IbEmergencyStop,
    bEstopAndDoors := IbEmergencyStop,
    bRun := VIS.bPucksInserterRun,
    bSimualtionMode := VIS.bSimulation,
    bHoming := bPucksInserterDoHoming OR btestHomingPI,
    bHeightSet := VIS.bPucksInserterHeightSet,
    bReset := PucksInserterError.bReset,
    bResetCycle := bCycleReseting,
    bIgnoreError := VIS.bPucksInserterIgnoreError,
    bSensorGate1On := IbPucksInserterGate1OnSensor,
    bSensorGate1Off := IbPucksInserterGate1OffSensor,
    bSensorGate2On := IbPucksInserterGate2OnSensor,
    bSensorGate2Off := IbPucksInserterGate2OffSensor,
    bSensorTrayOn := IbPucksInserterTrayOnSensor,
    bSensorTrayOff := IbPucksInserterTrayOffSensor,
    bSensorHammerUp := IbPucksInserterHammerUpSensor,
    bSensorHammerDown := IbPucksInserterHammerDownSensor,
    bSensorFormPositioningOn := IbPucksInserterFormPositioningOnSensor,
    bSensorFormPositioningOff := IbPucksInserterFormPositioningOffSensor,
    bSensorEntrySensor := IbPucksInserterWheelEntrySensor AND NOT VIS.bWeighingForm AND NOT VIS.bConfectionEnding,
    bSensorExitSensor := IbPucksInserterWheelExitSensor,
    bSensorFormPresent := IbPucksInserterFormGateBeforeSensor,
    bSensorFormAfterPresent := IbPucksInserterFormGateAfterSensor,
    bSensorHoming := IbPucksInserterHomingSensor,
    bSensorLevel := IbPucksInserterLevelSensor,
    bManualMovement := bManualMode,
    iStationIndex := 67,
    sStationName := 'Podajnik opakowań',
    tSensorBottleDelay := INT_TO_TIME(iPucksInserterBottleSensorDelay),
    tSensorFormDelay := INT_TO_TIME(iPucksInserterFormGateDelay+iPucksInserterFormGateDelayAdd),
    tAllowFormDelay := INT_TO_TIME(iPucksInserterAllowFormDelay),
    lrHammerHeightSV := lrPucksInserterHammerHeightSV,
    udiHeightMotorEncoderCV := IudiPucksInserterHammerHeightEncoderCV,
    bHeightEncoderSetCDone := IbPucksInserterHammerHeightEncoderSetCDone,
    rHeightMotorPositionOffset := 323,
    lrMaxHeight := 323,
    lrMinHeight := 80,
    bConveyorOK := IbPucksInserterTransporter2OK,
    InConveyorVelocityCV := uiPucksInserterConveyorActualVelocity,
    InConveyorSTW := uiPucksInserterConveyorSW,
    IbConveyorWcState := IbPucksInserterConveyorWcState,
    udiConveyorVelocitySV := iPucksInserterConveyorVelocitySV,
    iWheelSlots := 8,
    IiWheelZPhaseOffset := diPucksInserterWheelZPhaseOffset,
    lrWheelOffset := lrPucksInserterWheelOffset,
    lrWheelAcceleration := lrPucksInserterWheelAcceleration,
    lrWheelDeceleration := lrPucksInserterWheelAcceleration,
    lrWheelJerk := 100000,
    lrWheelVelocity := lrPucksInserterWheelVelocity,
    _MANUAL_ := bTest2,
    bManualHammer := VIS.bPucksInserterManualHammer,
    bManualHeightMotorUp := VIS.bPucksInserterManualHammerUp,
    bManualHeightMotorDown := VIS.bPucksInserterManualHammerDown,
    bManuaTray := VIS.bPucksInserterManualTray,
    bManualGate1 := VIS.bPucksInserterManualGate1,
    bManualGate2 := VIS.bPucksInserterManualGate2,
    bManualFormPositioning := VIS.bPucksInserterManualFormPositioning,
    bManualConveyor := VIS.bPucksInserterConveyorManualCmdStart,
    bManualWheelLeft := VIS.bPucksInserterManualWheelLeft,
    bManualWheelRight := VIS.bPucksInserterManualWheelRight,
    WheelAxisRef := aPucksInserterWheelAxisRef,
    eRunningState => ePucksInserterRunningState,
    bError => PucksInserterError.bError,
    udiErrorID => PucksInserterError.nErrorCode,
    sErrorDescription => PucksInserterError.sErrorString,
    sErrorDescription2 => PucksInserterError.sErrorString2,
    udiStationID => PucksInserterError.udiStationID,
    sErrorStationName => PucksInserterError.sStationName,
    bHeightMotorUp => QbPucksInserterHammerHeightUpCmd,
    bHeightMotorDown => QbPucksInserterHammerHeightDownCmd,
    udiHeightMotorEncoderSetCV => QudiPucksInserterHammerHeightEncoderSetCV,
    bHeightEncoderSetC => QbPucksInserterHammerHeightEncoderSetC,
    lrHeightMotorCV => VIS.lrPucksInserterHammerHeightCV,
    QnConveyorVelocitySV => udiPucksInserterConveyorVelocity,
    QnConveyorCTW => uiPucksInserterConveyorCW,
    lrWheelPositionCV => VIS.lrPucksInserterWheelPositionCV,
    bHammer => QbPucksInserterHammer,
    bTray => QbPucksInserterTray,
    bGate1 => QbPucksInserterGate1,
    bGate2 => QbPucksInserterGate2,
    bFormPositioning => QbPucksInserterFormPositioning); // FB_PucksInserter
ePucksInserterStationState := fbPucksInserter.eState;
END_ACTION

ACTION aPushTable:
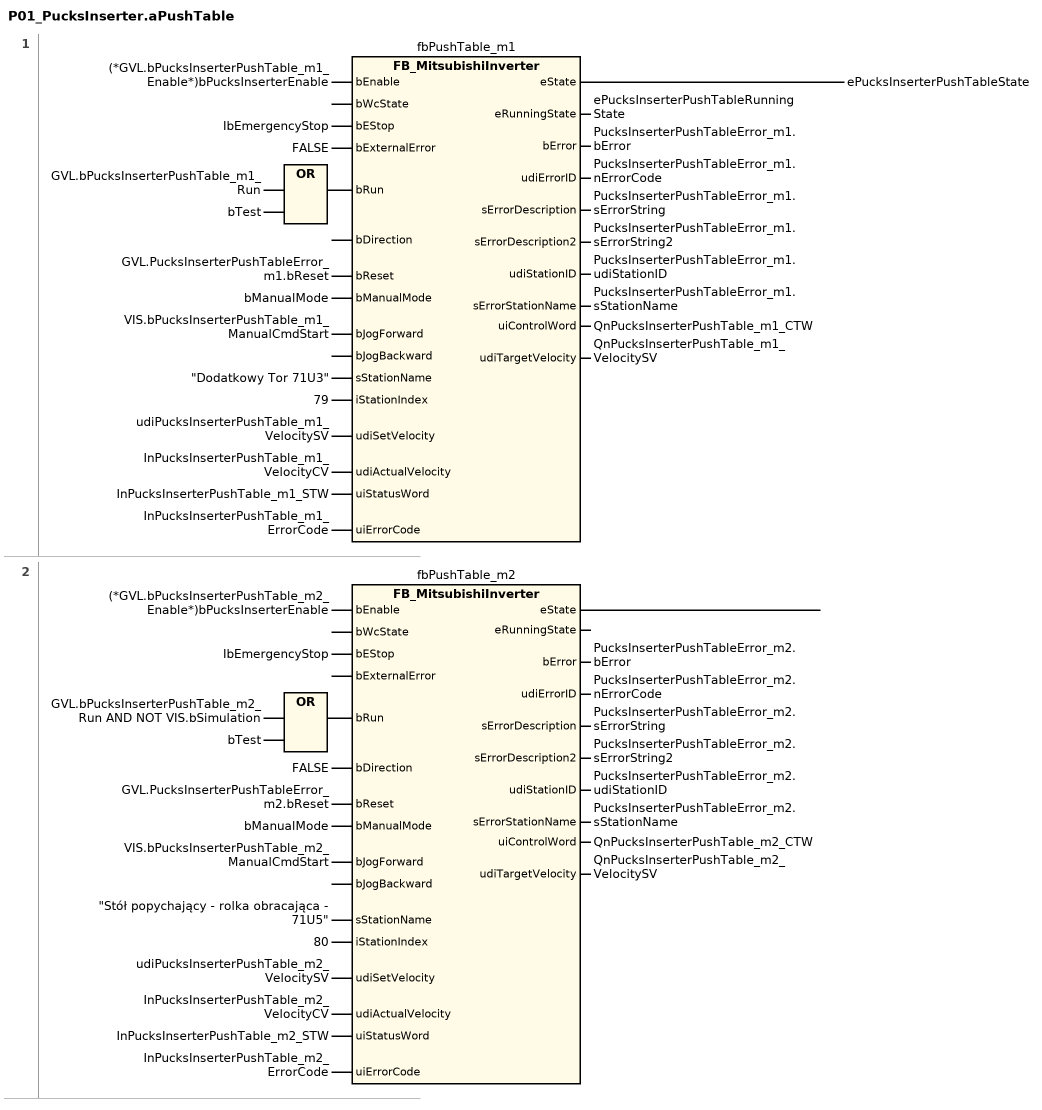
// NETWORK 1
fbPushTable_m1(
    bEnable := (*GVL.bPucksInserterPushTable_m1_Enable*)bPucksInserterEnable,
    bEStop := IbEmergencyStop,
    bExternalError := FALSE,
    bRun := GVL.bPucksInserterPushTable_m1_Run OR bTest,
    bReset := GVL.PucksInserterPushTableError_m1.bReset,
    bManualMode := bManualMode,
    bJogForward := VIS.bPucksInserterPushTable_m1_ManualCmdStart,
    sStationName := "Dodatkowy Tor 71U3",
    iStationIndex := 79,
    udiSetVelocity := udiPucksInserterPushTable_m1_VelocitySV,
    udiActualVelocity := InPucksInserterPushTable_m1_VelocityCV,
    uiStatusWord := InPucksInserterPushTable_m1_STW,
    uiErrorCode := InPucksInserterPushTable_m1_ErrorCode,
    eRunningState => ePucksInserterPushTableRunningState,
    bError => PucksInserterPushTableError_m1.bError,
    udiErrorID => PucksInserterPushTableError_m1.nErrorCode,
    sErrorDescription => PucksInserterPushTableError_m1.sErrorString,
    sErrorDescription2 => PucksInserterPushTableError_m1.sErrorString2,
    udiStationID => PucksInserterPushTableError_m1.udiStationID,
    sErrorStationName => PucksInserterPushTableError_m1.sStationName,
    uiControlWord => QnPucksInserterPushTable_m1_CTW,
    udiTargetVelocity => QnPucksInserterPushTable_m1_VelocitySV); // FB_MitsubishiInverter
ePucksInserterPushTableState := fbPushTable_m1.eState;

// NETWORK 2
fbPushTable_m2(
    bEnable := (*GVL.bPucksInserterPushTable_m2_Enable*)bPucksInserterEnable,
    bEStop := IbEmergencyStop,
    bRun := (GVL.bPucksInserterPushTable_m2_Run AND NOT VIS.bSimulation) OR bTest,
    bDirection := FALSE,
    bReset := GVL.PucksInserterPushTableError_m2.bReset,
    bManualMode := bManualMode,
    bJogForward := VIS.bPucksInserterPushTable_m2_ManualCmdStart,
    sStationName := "Stół popychający - rolka obracająca - 71U5",
    iStationIndex := 80,
    udiSetVelocity := udiPucksInserterPushTable_m2_VelocitySV,
    udiActualVelocity := InPucksInserterPushTable_m2_VelocityCV,
    uiStatusWord := InPucksInserterPushTable_m2_STW,
    uiErrorCode := InPucksInserterPushTable_m2_ErrorCode,
    bError => PucksInserterPushTableError_m2.bError,
    udiErrorID => PucksInserterPushTableError_m2.nErrorCode,
    sErrorDescription => PucksInserterPushTableError_m2.sErrorString,
    sErrorDescription2 => PucksInserterPushTableError_m2.sErrorString2,
    udiStationID => PucksInserterPushTableError_m2.udiStationID,
    sErrorStationName => PucksInserterPushTableError_m2.sStationName,
    uiControlWord => QnPucksInserterPushTable_m2_CTW,
    udiTargetVelocity => QnPucksInserterPushTable_m2_VelocitySV); // FB_MitsubishiInverter

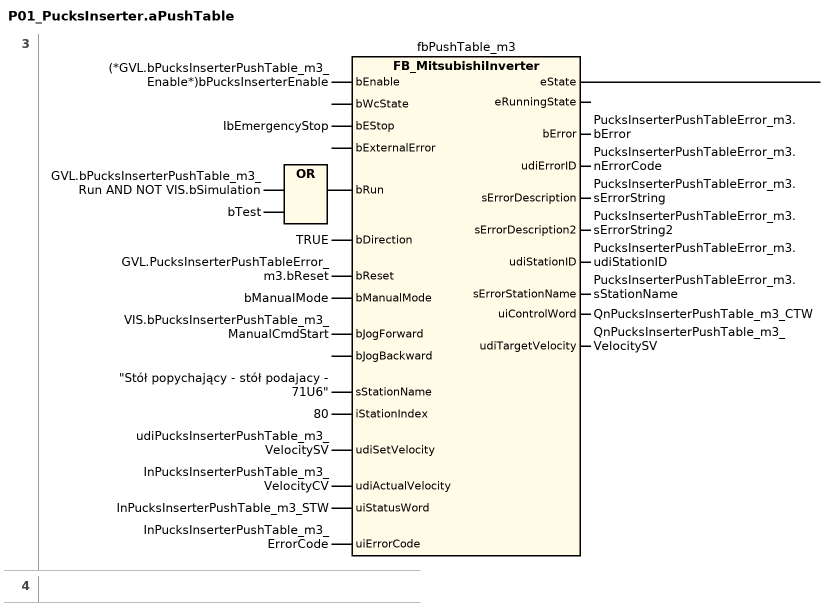
// NETWORK 3
fbPushTable_m3(
    bEnable := (*GVL.bPucksInserterPushTable_m3_Enable*)bPucksInserterEnable,
    bEStop := IbEmergencyStop,
    bRun := (GVL.bPucksInserterPushTable_m3_Run AND NOT VIS.bSimulation) OR bTest,
    bDirection := TRUE,
    bReset := GVL.PucksInserterPushTableError_m3.bReset,
    bManualMode := bManualMode,
    bJogForward := VIS.bPucksInserterPushTable_m3_ManualCmdStart,
    sStationName := "Stół popychający - stół podajacy - 71U6",
    iStationIndex := 80,
    udiSetVelocity := udiPucksInserterPushTable_m3_VelocitySV,
    udiActualVelocity := InPucksInserterPushTable_m3_VelocityCV,
    uiStatusWord := InPucksInserterPushTable_m3_STW,
    uiErrorCode := InPucksInserterPushTable_m3_ErrorCode,
    bError => PucksInserterPushTableError_m3.bError,
    udiErrorID => PucksInserterPushTableError_m3.nErrorCode,
    sErrorDescription => PucksInserterPushTableError_m3.sErrorString,
    sErrorDescription2 => PucksInserterPushTableError_m3.sErrorString2,
    udiStationID => PucksInserterPushTableError_m3.udiStationID,
    sErrorStationName => PucksInserterPushTableError_m3.sStationName,
    uiControlWord => QnPucksInserterPushTable_m3_CTW,
    udiTargetVelocity => QnPucksInserterPushTable_m3_VelocitySV); // FB_MitsubishiInverter

// NETWORK 4
END_ACTION

ACTION aTurntable:
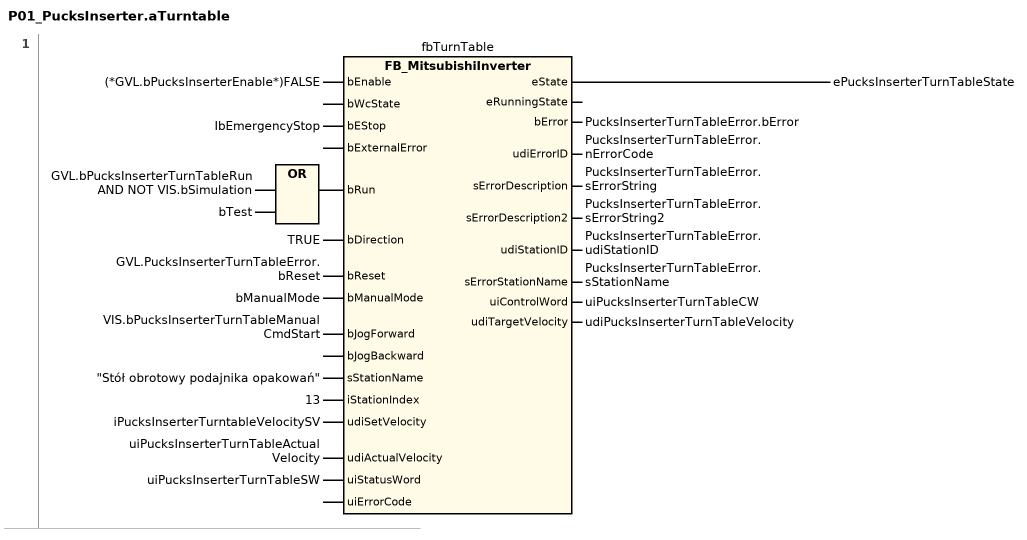
// NETWORK 1
fbTurnTable(
    bEnable := (*GVL.bPucksInserterEnable*)FALSE,
    bEStop := IbEmergencyStop,
    bRun := (GVL.bPucksInserterTurnTableRun AND NOT VIS.bSimulation) OR bTest,
    bDirection := TRUE,
    bReset := GVL.PucksInserterTurnTableError.bReset,
    bManualMode := bManualMode,
    bJogForward := VIS.bPucksInserterTurnTableManualCmdStart,
    sStationName := "Stół obrotowy podajnika opakowań",
    iStationIndex := 13,
    udiSetVelocity := iPucksInserterTurntableVelocitySV,
    udiActualVelocity := uiPucksInserterTurnTableActualVelocity,
    uiStatusWord := uiPucksInserterTurnTableSW,
    bError => PucksInserterTurnTableError.bError,
    udiErrorID => PucksInserterTurnTableError.nErrorCode,
    sErrorDescription => PucksInserterTurnTableError.sErrorString,
    sErrorDescription2 => PucksInserterTurnTableError.sErrorString2,
    udiStationID => PucksInserterTurnTableError.udiStationID,
    sErrorStationName => PucksInserterTurnTableError.sStationName,
    uiControlWord => uiPucksInserterTurnTableCW,
    udiTargetVelocity => udiPucksInserterTurnTableVelocity); // FB_MitsubishiInverter
ePucksInserterTurnTableState := fbTurnTable.eState;
END_ACTION

ACTION aWarning:
// Warning 1
IF (IbBottleFeederSafetyDoor3Open AND bPucksInserterEnable) AND NOT BottleFeederWarning[0].bWarning THEN
	BottleFeederWarning[0].bWarning										:=TRUE;
	BottleFeederWarning[0].udiWarningCode								:=1;
	BottleFeederWarning[0].sDescription									:='Podajnik butelek | Otwarte drzwi dostępowe';
ELSIF (NOT GVL_io.IbBottleFeederSafetyDoor3Open OR NOT bPucksInserterEnable) (*AND PucksInserterWarning[0].bAcknowledge*) THEN
	BottleFeederWarning[0].bWarning										:= FALSE;
	BottleFeederWarning[0].bAcknowledge									:= FALSE;
	VIS.uliWarningAcknowledge.23 										:= FALSE;
//ELSIF PucksInserterWarning[0].bAcknowledge THEN
//ELSE
//	PucksInserterWarning[0].bAcknowledge									:= TRUE;
END_IF	

// Warning 2

IF (fbPucksInserter.bWarning1 AND bPucksInserterEnable) AND NOT BottleFeederWarning[1].bWarning THEN
	BottleFeederWarning[1].bWarning										:= TRUE;
	BottleFeederWarning[1].udiWarningCode								:= 2;
	BottleFeederWarning[1].sDescription									:= 'Podajnik butelek | Niski poziom butelek';
ELSIF (NOT fbPucksInserter.bWarning1 OR NOT bPucksInserterEnable) (*AND BottleFeederWarning[1].bAcknowledge*) THEN
	BottleFeederWarning[1].bWarning										:= FALSE;
	BottleFeederWarning[1].bAcknowledge									:= FALSE;
	VIS.uliWarningAcknowledge.26 										:= FALSE;
ELSIF BottleFeederWarning[1].bAcknowledge THEN
	BottleFeederWarning[1].bAcknowledge									:= TRUE;
END_IF

//Warning 3
IF (IbBottleFeederSafetyDoor1Open AND bPucksInserterEnable) AND NOT BottleFeederWarning[2].bWarning THEN
	BottleFeederWarning[2].bWarning										:=TRUE;
	BottleFeederWarning[2].udiWarningCode								:=3;
	BottleFeederWarning[2].sDescription									:='Podajnik butelek | Otwarta bramka wjazdowa';
ELSIF (NOT IbBottleFeederSafetyDoor1Open OR NOT bPucksInserterEnable) (*AND BottleFeederWarning[2].bAcknowledge*) THEN
	BottleFeederWarning[2].bWarning										:= FALSE;
	BottleFeederWarning[2].bAcknowledge									:= FALSE;
	VIS.uliWarningAcknowledge.41 										:= FALSE;
//ELSIF BottleFeederWarning[2].bAcknowledge THEN
//	BottleFeederWarning[2].bAcknowledge									:= TRUE;
END_IF	

//Warning 4
BottleFeederWarning[3].sDescription										:='Podajnik butelek | Otwarta bramka wyjazdowa';
IF (IbBottleFeederSafetyDoor2Open AND bPucksInserterEnable) AND NOT BottleFeederWarning[3].bWarning THEN
	BottleFeederWarning[3].bWarning										:=TRUE;
	BottleFeederWarning[3].udiWarningCode								:=4;
	BottleFeederWarning[3].sDescription									:='Podajnik butelek | Otwarta bramka wyjazdowa';
ELSIF (NOT GVL_io.IbBottleFeederSafetyDoor2Open OR NOT bPucksInserterEnable) (*AND BottleFeederWarning[3].bAcknowledge*) THEN
	BottleFeederWarning[3].bWarning										:= FALSE;
	BottleFeederWarning[3].bAcknowledge									:= FALSE;
	VIS.uliWarningAcknowledge.42 										:= FALSE;
//ELSIF BottleFeederWarning[3].bAcknowledge THEN
//	BottleFeederWarning[3].bAcknowledge									:= TRUE;
END_IF
END_ACTION

END_PROGRAM

// ---- POUs/FB/NewFBs/FB_PucksInserter.TcPOU
(*
Nazwa:	FB_PuckInserter
Opis:	Podajnik 
Wersja:	V0.12
Data:	13.01.2026
Autor:	DP
Urządzenia:	Szlabany docisku opakowań, pneumatyczne podnoszenie opakowań, szlabany formatki
Konfiguracja:	
Info:
Zmiany:
- [13.01.2026] Running w Manualu
- [dd.mm.rrrr] opis

*)

FUNCTION_BLOCK FB_PucksInserter
VAR_INPUT
	bEnable						: BOOL;					// Załączenie stacji 
	bEstop						: BOOL;					// Stop awaryjny
	bEstopAndDoors				: BOOL;					// Drzwi zamknięte	
	bRun						: BOOL;					// Rozkaz pracy
	bRunPrepare					: BOOL;					// Przygotowanie do rozpoczecia pracy
	bSimualtionMode				: BOOL;					// Bit od symulacji czujnika butelki 
	bHoming						: BOOL;					// Bazowanie stacji 
	bHeightSet					: BOOL;					// Ustawianie stacji 
	bReset						: BOOL;					// Resetowanie błędów stacji
	bResetCycle					: BOOL;					// Reset cyklu 
	bIgnoreError				: BOOL;					// Ignorowanie błędów
(**)bSensorGate1On				: BOOL;					// Czujnik siłownika szlabanu 1 / wysunięty
(**)bSensorGate1Off				: BOOL;					// Czujnik siłownika szlabanu 1 / wsunięty
(**)bSensorGate2On				: BOOL;					// Czujnik siłownika szlabanu 2 / wysunięty
(**)bSensorGate2Off				: BOOL;					// Czujnik siłownika szlabanu 2 / wsunięty
(**)bSensorTrayOn				: BOOL;					// Czujnik siłownika tacki / wysuniety
(**)bSensorTrayOff				: BOOL;					// Czujnik siłownika poziomego	/ wsunięty
(**)bSensorHammerUp				: BOOL;					// Czujnik siłownika wbijaka / góra
(**)bSensorHammerDown			: BOOL;					// Czujnik siłowniak wbijaka / dól
(**)bSensorFormPositioningOn	: BOOL;					// Czujnik pozycjonowania formatek wysunięty
(**)bSensorFormPositioningOff	: BOOL;					// Czujnik pozycjonowania formatek schowany
(**)bSensorEntrySensor			: BOOL;					// Czujnik obecności opakowania 
(**)bSensorExitSensor			: BOOL;					// Czujnik obecności opakowania 
(**)bSensorFormPresent			: BOOL;					// Czujnik obecności formatki
(**)bSensorFormAfterPresent		: BOOL;					// Czujnik obecności formatki za podajnikiem
(**)bSensorHoming				: BOOL;					// Czujnik bazowania serwa
(**)bSensorLevel				: BOOL;					// Czujnik poziomu

	bManualMovement				: BOOL;					// Zezwolenie na ręczne ruchy 	
	iStationIndex				: UDINT;				// Indywidualny numer stacji
	sStationName				: STRING;				// Nazwa stacji

	tSensorBottleDelay			: TIME;					// Czasówka na dojazd butelki na wejściu
	tSensorFormDelay			: TIME;					// Czasówka na stabilizacje formatki pod podajnikiem
	tAllowFormDelay				: TIME;

	_HEIGHTMOTOR_ 				: BOOL;
	lrHammerHeightSV			: LREAL;				// Zadana wysokość
	udiHeightMotorEncoderCV		: UDINT;				// Ilość impulsów z modułu enkoderowego
	bHeightEncoderSetCDone		: BOOL;					// Zerowanie enkodera wykonane
	rHeightMotorPositionOffset 	: REAL;					// Wysokość bazowani podnośnika
	lrMaxHeight					: LREAL;				// Maksymalna wysokość podnośnika chwytaka
	lrMinHeight					: LREAL;				// Minimalna wysokość podnośnika chwytaka
 
 	_CONVEYOR_					: BOOL;
	bConveyorOK					: BOOL;					// Wejście czujnika zabezpieczenia silnika 
	InConveyorVelocityCV 		: UDINT;		
	InConveyorSTW 				: UINT; 				// Statusword transportera wejściowo wyjściowego
	IbConveyorWcState			: BOOL; 				// Statusword transportera wejściowo wyjściowego
	udiConveyorVelocitySV		: UDINT;

	_AXIS_						: BOOL;
	iWheelSlots					: INT;
	IiWheelZPhaseOffset			: DINT;
	lrWheelOffset				: LREAL;		
	lrWheelAcceleration			: LREAL;	
	lrWheelDeceleration			: LREAL;	
	lrWheelJerk					: LREAL;	
	lrWheelVelocity				: LREAL;		
END_VAR

VAR_OUTPUT
	                     
	eState						: E_Station;
	eRunningState				: E_PuckInserterState;	// Stan przeciągania formatek
	bError						: BOOL;					// Błąd stacji
	udiErrorID					: UDINT;				// Nr blędu przeciągania formatek
	sErrorDescription			: STRING(200);			// Opis błędu
	sErrorDescription2			: STRING(200);			// Opis błędu
	udiStationID				: UDINT;				// Nr stacji	
	sErrorStationName			: STRING;				// Nazwa stacji

	bHeightMotorUp				: BOOL;					//Sterowanie silnikiem podnośnika  - RUCH W GÓRĘ
	bHeightMotorDown			: BOOL;					//Sterowanie silnikiem podnośnika  - RUCH W DÓŁ
	udiHeightMotorEncoderSetCV	: UDINT;		
	bHeightEncoderSetC			: BOOL;					// Zerowanie enkodera
	lrHeightMotorCV				: LREAL;				// Aktualna pozycja podnośnika

	QnConveyorVelocitySV 		: UDINT; 				// Nastawa prędkości
	QnConveyorCTW 				: UINT;  				// Controlword transportera we/wy	
	lrWheelPositionCV			: LREAL;				// Aktualna pozycja karuzeli

	bHammer						: BOOL;					// Wbijak
	bTray						: BOOL;					// Tacka
	bGate1						: BOOL;					// Otwarcie szlabanu 1 / wysnięty (opakowania)							
	bGate2						: BOOL;					// Otwarcie szlabanu 2 / wysnięty (opakowania)				
	bFormPositioning			: BOOL;					// Pozycjonowanie formatek

	bCycleDone					: BOOL;					// Sygnał zakończenia cyklu
	bCycleNotDone				: BOOL;					// Sygnał błędnego zakończenia cyklu 
	bHomingDone					: BOOL;					// Sygnał zbazowania stacji 
	tCycleTime					: TIME;					// Czas syklu stacji 
	sWarning1Description		: STRING;
	bWarning1					: BOOL;
	sWarning2Description		: STRING;
	bWarning2					: BOOL;
	udiWarningID				: UDINT;	
	
	eRunningStateBeforeEstop	: E_PuckInserterState; 	// Stan przed Estope
	
END_VAR

VAR_IN_OUT
	
	_MANUAL_					: BOOL;	
	bManualHammer				: BOOL;					// Wbijak
	bManualHeightMotorUp		: BOOL;					// W góre
	bManualHeightMotorDown		: BOOL;					// W dół
	bManuaTray					: BOOL;					// Lewo
	bManualGate1				: BOOL;					// Szlaban 1 - lewy
	bManualGate2				: BOOL;					// Szlaban 2 - lewy
	bManualFormPositioning		: BOOL;					// Pozycjonowanie formatki
	bManualConveyor				: BOOL; 				// Start transportera		
	bManualWheelLeft 			: BOOL; 				// Karuzela - przód		
	bManualWheelRight 			: BOOL; 				// Karuzela - tył		
	WheelAxisRef				: AXIS_REF;		

END_VAR

VAR
	// State
	eLastState									: E_Station;						//Stan ogólny bloku
	eLastStateTemp								: E_Station;						//Stan ogólny bloku
	eLastRunningState							: E_PuckInserterState;				//Stan podbloku
	eLastRunningStateTemp						: E_PuckInserterState;				//Stan podbloku
	
	bHammerLastState							: BOOL;
	bTrayLastState								: BOOL;	
	bGate1LastState								: BOOL;			
	bGate2LastState								: BOOL;				
	bFormPositioningLastState					: BOOL;

	//Axis online
	fbWheel										: FB_McAxisOnlineNC;
	stWheel										: ST_McAxisOnline;
	lrWheelOffsetWhenHoming						: LREAL;
	lrWheelLastKnownPosition					: LREAL;	
	
	//Inverter
	fbConveyor									: FB_MitsubishiInverter;
	
	//Reset 
	rtResetCycle: R_TRIG;			
	rtrigCycleTimerRead							: R_TRIG;							// Do zliczania czasu
	tonCycleTimer								: TON;								// Timer
	bResetCycleOn								: BOOL;

	//Triggery
	ftIbSensorHammerDown						: F_TRIG;							// Triger zjazdu z dolnego czujnika
	rtResetCommands								: R_TRIG;
	tonfbConveyorbRun							: TON;
	// czasówki
	tonPreparingToDisabled						: TON;								// Czasówka za długiego przygotowania do gotowosic
	tonPreparingToReadyOn						: TON;								// Czasówka za długiego przygotowania do gotowosic
	tonBottleEntrySensorDelay					: TON;								// Czasówka na załączenie wykrycia butelki
	tonBottleExitSensorDelay					: TON;								// Czasówka na załączenie wykrycia butelki
	tonAllowEmptyForm							: TON;
	tonFormsPresentDelay						: TON;								// Czasówka na załączenie obecności formatki
	tonResetting								: TON;
	
	//czasówki od błędów	
	tonGate1OnError								: TON;
	tonGate1OffError							: TON;
	tonGate2OnError								: TON;
	tonGate2OffError							: TON;
	tonTrayOnError								: TON;
	tonTrayOffError								: TON;
	tonHammerOnError							: TON;
	tonHammerOffError							: TON;
	tonFormPositioningOnError					: TON;
	tonFormPositioningOffError					: TON;
	tonBottleAndFormTooLong						: TON;
	tonOpeningBlocked							: TON;
	tonErrorHeightChange						: TON; 	
	tonMaxHeight								: TON; 
	tonMinHeight								: TON; 	
	tonSVCVDiffHeight							: TON; 	
	
	// case
	iHomingStep									: INT;
	iAbortingCase								: INT;
	iPreparingToMoveCase						: INT;
	// bit bledow
	bStateError									: BOOL;
	bWasErrorOrEstop							: BOOL;
	
	//Warning
	fbLevelSensor								: FB_InputFilter_v2;

	bSimulationSensor							: BOOL;
	tonEstopDelay: TON;
	
	
	tonGripper: TON;
	tonOpenedGripper: TON;
	tofRunning: TOF;
	tonReady: TON;
	tonArmDown: TON;

	//Podnośnik Jiesang	
	fbHeightMotorEncoder: FB_JiesangActuatorEncoderModul;	//FB_JiesangActuatorEncoder;	// Blok enkodera podnośnika chwytaka stabilizującego pod zakręcarką	
	bHeightMotorEncoderCounterReset: BOOL; 					//Sygnał resetu enkodera
	bHeightMotorEncoderHomed: BOOL;							//Informacja od enkodera że jest zbazowany
	nLastPositionHeightCV: LREAL;							//Pozycja podnośnika w poprzednim cyklu programu
	tonLimitPosMinReachedDelay: TON;
	tonLimitPosMaxReachedDelay: TON;
	tonHeightNoChange: TON; 								//Timer wykrycia braku ruchu siłownika zmiany wysokości stacji
	rtEncoderHomed:R_TRIG;
	tofMotorUpPermition: TOF;
	tofMotorDownPermition: TOF;
	tofHeightMotorDown: TOF;
	
	iTurningTest:INT;
	bWheelOffsetChanged:BOOL;
	bWasEstop:BOOL;
	iPreparingToReadyCase:INT;
	
	//Zmienne od EVENTLOGGER
	bAlarmInit 						: BOOL := TRUE; 
	nAlarmNumerator					: INT;
	arfbAlarm						: ARRAY[0..19] OF  FB_TcAlarm;		//Tablica bloczków błędów
	fbSourceInfo 					: FB_TcSourceInfo;
	iSourceInfo						: I_TcSourceInfo;
	sAlarmTest						: STRING;
	//Koniec zmiennych od EVENTLOGGER
	
	
	
	tonWheelError: TON;
	lrTemp: LREAL;
END_VAR


aLimits();
aHeightMotor();
aWheelControlBlocks();
aErrorHandling();
aSignals();
aControl();
aInverter();
aStatistic();
aWarnings();
aStationID();
aCycleReset();
(*Zapisywanie ostatniego stanu*)
IF eLastStateTemp<>eState THEN
	eLastState := eLastStateTemp;
END_IF
eLastStateTemp := eState;
IF eLastRunningStateTemp<>eRunningState THEN
	eLastRunningState := eLastRunningStateTemp;
END_IF
eLastRunningStateTemp := eRunningState;
(*Koniec Zapisywanie ostatniego stanu*)

nLastPositionHeightCV:=lrHeightMotorCV;

ACTION aControl:

//Wyłączenie stacji
IF NOT bEnable THEN
	IF eState <> E_Station.eRunning AND eState <> E_Station.eDisabled AND eState <> E_Station.ePreparingToDisable THEN
		eState										:=	E_Station.ePreparingToDisable;
	END_IF
END_IF
	
// Praca po Estopie
IF NOT bEstop  THEN	
	IF eState <> E_Station.eAborted AND eState <> E_Station.eAborting AND eState <> E_Station.eDisabled THEN
			eRunningStateBeforeEStop				:=	eRunningState;
			eState 									:=	E_Station.eAborting; 
			iAbortingCase							:= 0; 
	END_IF
END_IF
	
CASE eState OF
//--------------------------------------------------------------------------------
	E_Station.eDisabled:
		IF bEnable THEN
			eState									:=	E_Station.ePreparingToReady;
		END_IF
	
//-------------------------------------------------------------------------------
	E_Station.ePreparingToDisable:
	
		stWheel.mcPower.bEnable						:= FALSE;
		stWheel.mcPower.bEnable_Negative			:= FALSE;
		stWheel.mcPower.bEnable_Positive			:= FALSE;
		stWheel.mcPower.lrOverride					:= 0;
		
		bWasErrorOrEstop							:= FALSE;
		bHomingDone									:= FALSE;	 

		bHammer										:= FALSE; 
		bTray										:= FALSE;
		bGate1										:= FALSE;			
		bGate2										:= FALSE;   			
		bFormPositioning							:= FALSE;  
		
		bHeightMotorUp								:= TRUE;
		bHeightMotorDown							:= FALSE;	
		
		IF tonHeightNoChange.Q THEN
			bHeightMotorUp							:=	FALSE;
			IF NOT stWheel.mcPower.bStatus THEN
				aResetCommands();
				eState								:=	E_Station.eDisabled;
				eRunningState						:=	E_PuckInserterState.eDisabled;
			END_IF
		END_IF	

//--------------------------------------------------------------------------------
	E_Station.eAborted:
		IF bEstop THEN
			bWasErrorOrEstop						:= TRUE;	
			eState									:= E_Station.ePreparingToReady;
		END_IF

//--------------------------------------------------------------------------------	
	E_Station.eAborting:
	
		IF NOT bEstop THEN
			bWasEstop	:= 	TRUE;
		END_IF
	
		CASE iAbortingCase OF
			
			0: //Inicjalizacja
				IF stWheel.mcPower.bStatus THEN
					iAbortingCase					:= 10;
				ELSE
					iAbortingCase					:= 40;
				END_IF
				
			10: //Komenda MC_STOP
				stWheel.mcStop.bExecute				:= TRUE;	
				//Czekam na Done
				IF stWheel.mcStop.bDone THEN
					stWheel.mcStop.bExecute			:= FALSE;
					iAbortingCase					:= 20;
				END_IF
				
			20: //Kasowanie komend
				stWheel.mcMoveAbsolute.bExecute		:= FALSE;
				stWheel.mcMoveRelative.bExecute		:= FALSE;
				aResetCommandsNoTray();
				iAbortingCase						:= 30;
	
			30: //Wyłączenie osi
				stWheel.mcPower.bEnable				:= FALSE;
				stWheel.mcPower.bEnable_Negative	:= FALSE;
				stWheel.mcPower.bEnable_Positive	:= FALSE;
				IF NOT stWheel.mcPower.bStatus THEN
					iAbortingCase					:= 40;
				END_IF
				
			40: //Kasowanie podzespołow
				aResetCommandsNoTray();
				iAbortingCase						:= 50;
				
			50: //Przejście do Aborted
				iAbortingCase						:= 0;
				eState								:= E_Station.eAborted;
				eRunningState						:= E_PuckInserterState.eDisabled;
				
		END_CASE
		
//--------------------------------------------------------------------------------
	E_Station.eError:
	
		bWasErrorOrEstop							:= TRUE;
		IF bReset THEN
			eState									:= E_Station.eResetting;
			bError									:= FALSE;
		ELSE
			aResetCommands();	
		END_IF

//--------------------------------------------------------------------------------
	E_Station.eResetting:

				bTray								:= FALSE;

				bHammer								:= FALSE; 	

				stWheel.mcReset.bExecute			:= TRUE;
				fbConveyor.bReset					:= TRUE;
				IF NOT fbConveyor.bError AND stWheel.mcReset.bDone THEN
					stWheel.mcReset.bExecute		:= FALSE;
					fbConveyor.bReset				:= FALSE;
					bError							:= FALSE;
				END_IF				

					

	
		IF NOT bError AND fbConveyor.eState = E_Station.eReady THEN
			fbConveyor.bReset	:= FALSE;	
			udiErrorID								:= 0;
			sErrorDescription						:= '';
			sErrorDescription2						:= '';
			iPreparingToReadyCase					:=	0;
			eState									:= E_Station.ePreparingToReady;
		ELSIF tonResetting.Q THEN   //200ms                	
			eState									:= E_Station.eError;
		END_IF

//--------------------------------------------------------------------------------			
	E_Station.eManualMovement: 
		aManualMovements();
		IF NOT bManualMovement THEN
			bHeightMotorUp							:=	FALSE;
			bHeightMotorDown						:=	FALSE;
			bHammer									:=	bHammerLastState;			
			bTray									:=	bTrayLastState;				
			bGate1									:=	bGate1LastState;			
			bGate2									:=	bGate2LastState;				
			bFormPositioning						:=	bFormPositioningLastState;	
			eState									:=	E_Station.eReady;
		END_IF
		
//--------------------------------------------------------------------------------
	E_Station.eHoming: 			
		bHomingDone 								:= FALSE;
		aHoming();
		IF NOT bHoming AND NOT bHeightSet THEN 
		   	bHeightMotorDown						:= FALSE;
			bHeightMotorUp							:= FALSE;
			eState									:= E_Station.ePreparingToReady;
		END_IF

//--------------------------------------------------------------------------------	
	E_Station.eHomingDone:
	
//		fbHeightMotorEncoder.bHomingCancel			:= FALSE;
		bHeightMotorDown							:=	FALSE;
		bHeightMotorUp								:=	FALSE;
		bHeightMotorEncoderCounterReset				:=	FALSE;	
		bHomingDone									:=	TRUE;
		IF NOT bHoming	AND NOT bHeightSet THEN
			eState									:= E_Station.ePreparingToReady;
		END_IF

//--------------------------------------------------------------------------------				
	E_Station.ePreparingToReady:

	//bWasEstop;
	CASE iPreparingToReadyCase OF
		
		0:
			IF tonPreparingtoReadyOn.Q THEN
			
				stWheel.mcPower.bEnable					:= TRUE;
				stWheel.mcPower.bEnable_Negative		:= TRUE;
				stWheel.mcPower.bEnable_Positive		:= TRUE;
				stWheel.mcPower.lrOverride				:= 100;
                                                                                          
				IF stWheel.mcPower.bStatus  AND NOT stWheel.bError THEN     
//				  iPreparingToReadyCase	:=	100;
//				ELSE
					iPreparingToReadyCase	:=	iPreparingToReadyCase	+	5;
				END_IF
			END_IF	
		5:
					 iPreparingToReadyCase			:=	10;			
		10:
				stWheel.mcReset.bExecute			:= TRUE;
				IF stWheel.mcReset.bDone THEN
					stWheel.mcReset.bExecute		:= FALSE;
				END_IF	
				IF  NOT stWheel.bError   THEN   
					 iPreparingToReadyCase			:=	15;
				END_IF
		15:
				IF tonPreparingToReadyOn.Q THEN
					 iPreparingToReadyCase			:=	20;
				ELSIF NOT bHomingDone THEN
					 iPreparingToReadyCase			:=	100;
		
				END_IF	
		20:
		
		IF  (
					(ABS(LMOD(WheelAxisRef.NcToPlc.ModuloActPos,360.0/iWheelSlots)) > (360.0/iWheelSlots*0.01)) AND
					(ABS(LMOD(WheelAxisRef.NcToPlc.ModuloActPos,360.0/iWheelSlots)) < (360.0/iWheelSlots*0.99))  
					)
					AND NOT (LMOD(WheelAxisRef.NcToPlc.ModuloActPos,360.0/iWheelSlots) = 0) 
					THEN                    
						lrTemp := LMOD(WheelAxisRef.NcToPlc.ModuloActPos,360.0/iWheelSlots);   
						 stWheel.mcMoveModulo.lrPosition	:=	(WheelAxisRef.NcToPlc.ModuloActPos+360.0/iWheelSlots-LMOD(WheelAxisRef.NcToPlc.ModuloActPos,360.0/iWheelSlots))
						
						;
				ELSE
						stWheel.mcMoveModulo.lrPosition	:=	WheelAxisRef.NcToPlc.ModuloActPos;				
				END_IF 

					stWheel.mcMoveModulo.bExecute			:=	TRUE;
					stWheel.mcMoveModulo.lrVelocity		:=	lrWheelVelocity / 2;
					stWheel.mcMoveModulo.lrAcceleration	:=	lrWheelAcceleration / 2;
					stWheel.mcMoveModulo.lrDeceleration	:=	lrWheelDeceleration / 2;
					 iPreparingToReadyCase			:=	30;		
			30:						
					IF stWheel.mcMoveModulo.bDone THEN	
						stWheel.mcMoveModulo.bExecute		:=	FALSE;
						iPreparingToReadyCase := 100;
					END_IF
		100:
		
				aResetCommandsNoTray();                  
				bWasEstop							:= FALSE;
				eState								:= E_Station.eReady;
				eRunningState						:= E_PuckInserterState.eReady;
				IF bResetCycleOn THEN               
					eState							:= E_Station.eHoming;
				END_IF				
	
	END_CASE


//--------------------------------------------------------------------------------
// Stan gotowości
		
	E_Station.eReady:
		
		IF tonReady.Q THEN
			fbConveyor.bRun 							:= FALSE;
		END_IF
		
		//IF rtResetCommands.Q THEN	aResetCommands();	END_IF		
		
		IF bRunPrepare OR bRun AND (NOT bCycleDone AND NOT bCycleNotDone) THEN
			eState									:= E_Station.eStarting;
		END_IF
		
		IF bHoming OR bHeightSet THEN
			eState									:= E_Station.eHoming;
		END_IF
		
		IF bManualMovement THEN	
			bManualHammer							:=	bHammerLastState			:= bHammer;	
			bManualHeightMotorUp					:=	bHeightMotorUp;
			bManualHeightMotorDown					:=	bHeightMotorDown;
			bManuaTray								:=  bTrayLastState				:= bTray;	
			bManualGate1							:=	bGate1LastState				:= bGate1;		
			bManualGate2							:=	bGate2LastState				:= bGate2;	
			bManualFormPositioning					:=  bFormPositioningLastState	:= bFormPositioning;	
			bManualConveyor							:=	FALSE;		
			bManualWheelLeft 						:=	FALSE;
			bManualWheelRight 						:=	FALSE;	
			eState									:=	E_Station.eManualMovement;
			eRunningState							:=	E_PuckInserterState.eReady;
		END_IF
		
		IF NOT bRun  THEN
			bCycleDone								:=	FALSE;
			bCycleNotDone 							:=	FALSE;
		END_IF

//--------------------------------------------------------------------------------
	E_Station.eStopping:
	
		aRunning();
		IF eRunningState =	E_PuckInserterState.eReady OR eRunningState	= E_PuckInserterState.ePreparingToMove  THEN
			eRunningState							:=	E_PuckInserterState.eReady;
			eState									:=	E_Station.eReady;
		END_IF
		IF eRunningState =	E_PuckInserterState.eGoAbove OR 
			(eRunningState =	E_PuckInserterState.eInsterting AND NOT bHammer) THEN
			eState									:=	E_Station.eReady;
		END_IF
		
//--------------------------------------------------------------------------------
	E_Station.eStarting:
	(*
			IF  (
				(ABS(LMOD(WheelAxisRef.NcToPlc.ActPos,360.0/iWheelSlots)) > (360.0/iWheelSlots*0.01)) AND
				(ABS(LMOD(WheelAxisRef.NcToPlc.ActPos,360.0/iWheelSlots)) < (360.0/iWheelSlots*0.99))  
				)
				AND NOT (LMOD(WheelAxisRef.NcToPlc.ActPos,360.0/iWheelSlots) = 0) 
				THEN                       
					 stWheel.mcMoveAbsolute.lrPosition	:=	(WheelAxisRef.NcToPlc.ActPos+360.0/iWheelSlots-LMOD(WheelAxisRef.NcToPlc.ActPos,360.0/iWheelSlots))
						
					;
			ELSE
					stWheel.mcMoveAbsolute.lrPosition	:=	WheelAxisRef.NcToPlc.ActPos;				
			END_IF 
				stWheel.mcMoveAbsolute.bExecute			:=	TRUE;
				stWheel.mcMoveAbsolute.lrVelocity		:=	lrWheelVelocity / 2;
				stWheel.mcMoveAbsolute.lrAcceleration	:=	lrWheelAcceleration / 2;
				stWheel.mcMoveAbsolute.lrDeceleration	:=	lrWheelDeceleration / 2;
					
				IF stWheel.mcMoveAbsolute.bDone THEN	
			    	stWheel.mcMoveAbsolute.bExecute		:=	FALSE;
					eState								:=	E_Station.eRunning;
			    END_IF	
		*)
		eState								:=	E_Station.eRunning;
//--------------------------------------------------------------------------------
	E_Station.eRunning:	
		
		aRunning();
		IF NOT bRun	THEN
			eState									:=	E_Station.eStopping;
		END_IF

		IF bCycleDone OR bCycleNotDone THEN (*Cykl zakończony*)
			eState									:=	E_Station.eReady;
		END_IF
		
END_CASE
END_ACTION

ACTION aCycleReset:

(*****Reset bloczka*****)
IF bEnable THEN
	IF eState <> E_Station.eDisabled AND eState <> E_Station.ePreparingToDisable THEN
		IF bResetCycle THEN
			bResetCycleOn						:= TRUE;
			eState								:= E_Station.ePreparingToReady;
		END_IF
	END_IF
END_IF


IF bResetCycleOn THEN
	
	aResetCommands();
	eRunningState							:= E_PuckInserterState.eReady;	
	eState 				 					:= E_Station.eReady;

END_IF
END_ACTION

ACTION aErrorHandling:
// Alarm_0520	520	Error	Blokada wysunięcia szlabanu 1 - lewy - odblokuj
// Alarm_0521	521	Error	Blokada schowania szlabanu 1 - lewy - odblokuj
// Alarm_0522	522	Error	Blokada wysunięcia szlabanu 2 - prawy - odblokuj
// Alarm_0523	523	Error	Blokada schowania szlabanu 2 - prawy - odblokuj
// Alarm_0524	524	Error	Blokada wysunięcia tacki - odblokuj
// Alarm_0525	525	Error	Blokada schowania tacki - odblokuj
// Alarm_0526	526	Error	Blokada opuszczania wbijaka - odblokuj
// Alarm_0527	527	Error	Blokada podnoszenia wbijaka - odblokuj
// Alarm_0528	528	Error	Blokada wysunięcia pozycjonowania formatek - odblokuj
// Alarm_0529	529	Error	Blokada schowania pozycjonowania formatek - odblokuj
// Alarm_0530	530	Error	Brak opakowań w podajniku - dołóż opakownia lub sprawdź ich ułożenie
// Alarm_0531	531	Error	Blokada podnośnika lub brak zasilania - sprawdź czujnik lub odblokuj mechanicznie
// Alarm_0532	532	Error	Wartość zadana wysokości jest większa od maksymalnej - zmień ustawienia w recepturze {0}
// Alarm_0533	533	Error	Wartość zadana wysokości jest mniejsza od minimalnej - zmień ustawienia w recepturze {0}
// Alarm_0534	534	Error	Wartość aktualna jest zbyt różna od zadanej - zmień ustawienia w recepturze lub ustaw stację
// Alarm_0535	535	Error	Błąd napędu karuzeli. Błąd NC: {0}
// Alarm_0536	536	Error	Błąd falownika przenośnika butelek: {0}


IF bAlarmInit THEN
    bAlarmInit := FALSE; 
	fbSourceInfo.Clear();
	fbSourceInfo.sName:=sLiteral_TO_UTF8(sStationName);
	fbSourceInfo.nId:=udiStationID;
	// Alarm_0520	520	Error	Blokada wysunięcia szlabanu 1 - lewy - odblokuj
    arfbAlarm[0].CreateEx(stEventEntry := TC_EVENTS.AlarmClass.Alarm_0520, bWithConfirmation:= FALSE,  ipSourceInfo:= fbSourceInfo); 
	// Alarm_0521	521	Error	Blokada schowania szlabanu 1 - lewy - odblokuj
	arfbAlarm[1].CreateEx(stEventEntry := TC_EVENTS.AlarmClass.Alarm_0521, bWithConfirmation:= FALSE,  ipSourceInfo:= fbSourceInfo); 
	// Alarm_0522	522	Error	Blokada wysunięcia szlabanu 2 - prawy - odblokuj
	arfbAlarm[2].CreateEx(stEventEntry := TC_EVENTS.AlarmClass.Alarm_0522, bWithConfirmation:= FALSE,  ipSourceInfo:= fbSourceInfo); 
	// Alarm_0523	523	Error	Blokada schowania szlabanu 2 - prawy - odblokuj
	arfbAlarm[3].CreateEx(stEventEntry := TC_EVENTS.AlarmClass.Alarm_0523, bWithConfirmation:= FALSE,  ipSourceInfo:= fbSourceInfo); 
	// Alarm_0524	524	Error	Blokada wysunięcia tacki - odblokuj
	arfbAlarm[4].CreateEx(stEventEntry := TC_EVENTS.AlarmClass.Alarm_0524, bWithConfirmation:= FALSE,  ipSourceInfo:= fbSourceInfo); 
	// Alarm_0525	525	Error	Blokada schowania tacki - odblokuj
	arfbAlarm[5].CreateEx(stEventEntry := TC_EVENTS.AlarmClass.Alarm_0525, bWithConfirmation:= FALSE,  ipSourceInfo:= fbSourceInfo); 
	// Alarm_0526	526	Error	Blokada opuszczania wbijaka - odblokuj
	arfbAlarm[6].CreateEx(stEventEntry := TC_EVENTS.AlarmClass.Alarm_0526, bWithConfirmation:= FALSE,  ipSourceInfo:= fbSourceInfo); 
	// Alarm_0527	527	Error	Blokada podnoszenia wbijaka - odblokuj
	arfbAlarm[7].CreateEx(stEventEntry := TC_EVENTS.AlarmClass.Alarm_0527, bWithConfirmation:= FALSE,  ipSourceInfo:= fbSourceInfo); 
	// Alarm_0528	528	Error	Blokada wysunięcia pozycjonowania formatek - odblokuj
	arfbAlarm[8].CreateEx(stEventEntry := TC_EVENTS.AlarmClass.Alarm_0528, bWithConfirmation:= FALSE,  ipSourceInfo:= fbSourceInfo); 
	// Alarm_0529	529	Error	Blokada schowania pozycjonowania formatek - odblokuj
	arfbAlarm[9].CreateEx(stEventEntry := TC_EVENTS.AlarmClass.Alarm_0529, bWithConfirmation:= FALSE,  ipSourceInfo:= fbSourceInfo); 
	// Alarm_0530	530	Error	Brak opakowań w podajniku - dołóż opakownia lub sprawdź ich ułożenie
	arfbAlarm[10].CreateEx(stEventEntry := TC_EVENTS.AlarmClass.Alarm_0530, bWithConfirmation:= FALSE,  ipSourceInfo:= fbSourceInfo); 
	// Alarm_0531	531	Error	Blokada podnośnika lub brak zasilania - sprawdź czujnik lub odblokuj mechanicznie
	arfbAlarm[11].CreateEx(stEventEntry := TC_EVENTS.AlarmClass.Alarm_0531, bWithConfirmation:= FALSE,  ipSourceInfo:= fbSourceInfo); 
	// Alarm_0532	532	Error	Wartość zadana wysokości jest większa od maksymalnej - zmień ustawienia w recepturze {0}
	arfbAlarm[12].CreateEx(stEventEntry := TC_EVENTS.AlarmClass.Alarm_0532, bWithConfirmation:= FALSE,  ipSourceInfo:= fbSourceInfo); 
	// Alarm_0533	533	Error	Wartość zadana wysokości jest mniejsza od minimalnej - zmień ustawienia w recepturze {0}
	arfbAlarm[13].CreateEx(stEventEntry := TC_EVENTS.AlarmClass.Alarm_0533, bWithConfirmation:= FALSE,  ipSourceInfo:= fbSourceInfo); 
	// Alarm_0534	534	Error	Wartość aktualna jest zbyt różna od zadanej - zmień ustawienia w recepturze lub ustaw stację
	arfbAlarm[14].CreateEx(stEventEntry := TC_EVENTS.AlarmClass.Alarm_0534, bWithConfirmation:= FALSE,  ipSourceInfo:= fbSourceInfo); 
	// Alarm_0535	535	Error	Błąd napędu karuzeli. Błąd NC: {0}
	arfbAlarm[15].CreateEx(stEventEntry := TC_EVENTS.AlarmClass.Alarm_0535, bWithConfirmation:= FALSE,  ipSourceInfo:= fbSourceInfo); 
	//Alarm_0536	536	Error	Błąd falownika przenośnika butelek: {0}
	arfbAlarm[16].CreateEx(stEventEntry := TC_EVENTS.AlarmClass.Alarm_0536, bWithConfirmation:= FALSE,  ipSourceInfo:= fbSourceInfo); 
END_IF




tonGate1OnError				(IN:= NOT bSensorGate1On				AND bGate1 								AND NOT bError, PT:=T#2S);
tonGate1OffError			(IN:= NOT bSensorGate1Off				AND NOT bGate1 							AND NOT bError, PT:=T#2S);
tonGate2OnError				(IN:= NOT bSensorGate2On				AND bGate2 								AND NOT bError, PT:=T#2S);
tonGate2OffError			(IN:= NOT bSensorGate2Off				AND NOT bGate2 							AND NOT bError, PT:=T#2S);
tonTrayOnError				(IN:= NOT bSensorTrayOn					AND bTray								AND NOT bError, PT:=T#2S);
tonTrayOffError				(IN:= NOT bSensorTrayOff				AND NOT bTray 							AND NOT bError, PT:=T#2S);
tonHammerOnError			(IN:= NOT bSensorHammerDown				AND bHammer								AND NOT bError AND NOT bManualMovement, PT:=T#2S);
tonHammerOffError			(IN:= NOT bSensorHammerUp				AND NOT bHammer 						AND NOT bError, PT:=T#2S);
//PI-usuniety bład do testów
//tonFormPositioningOnError	(IN:= NOT bSensorFormPositioningOn		AND bFormPositioning					AND NOT bError, PT:=T#2S); 
tonFormPositioningOffError	(IN:= NOT bSensorFormPositioningOff		AND NOT bFormPositioning 				AND NOT bError, PT:=T#2S);
//tonBottleAndFormTooLong		(IN:= NOT bSensorEntrySensor			AND NOT bError							AND bRun AND NOT bSimualtionMode, PT:=T#5M);//było 30s
tonEstopDelay				(IN:= bEStop,	PT:=T#3S);
bStateError					:= (eState = E_Station.eError OR eState = E_Station.eResetting);
	
IF (bEnable OR ((eState = E_Station.ePreparingToDisable) )) AND tonEstopDelay.Q THEN //AND NOT bError
	// Alarm_0520	520	Error	Blokada wysunięcia szlabanu 1 - lewy - odblokuj
	IF tonGate1OnError.Q THEN
		IF NOT arfbAlarm[0].bActive THEN
			arfbAlarm[0].Raise(nTimeStamp:=0);
		END_IF
	ELSE	
		IF  arfbAlarm[0].bActive AND bReset THEN
			arfbAlarm[0].Clear(nTimeStamp:=0, bResetConfirmation:= FALSE);
		END_IF
// 		bError 								:=	TRUE;
// 		udiErrorID							:=	320;
// 		sErrorDescription					:=	'Blokada wysunięcia szlabanu 1 - lewy - odblokuj';	
// 		sErrorDescription2					:=	'';			
	END_IF;
	// Alarm_0521	521	Error	Blokada schowania szlabanu 1 - lewy - odblokuj
	IF tonGate1OffError.Q THEN
		IF NOT arfbAlarm[1].bActive THEN
			arfbAlarm[1].Raise(nTimeStamp:=0);
		END_IF
	ELSE	
		IF  arfbAlarm[1].bActive AND bReset THEN
			arfbAlarm[1].Clear(nTimeStamp:=0, bResetConfirmation:= FALSE);
		END_IF
// 		bError 								:=	TRUE;
// 		udiErrorID							:=	321;
// 		sErrorDescription					:=	'Blokada schowania szlabanu 1 - lewy - odblokuj';	
// 		sErrorDescription2					:=	'';			
	END_IF;
	// Alarm_0522	522	Error	Blokada wysunięcia szlabanu 2 - prawy - odblokuj

	IF tonGate2OnError.Q THEN
		IF NOT arfbAlarm[2].bActive THEN
			arfbAlarm[2].Raise(nTimeStamp:=0);
		END_IF
	ELSE	
		IF  arfbAlarm[2].bActive AND bReset THEN
			arfbAlarm[2].Clear(nTimeStamp:=0, bResetConfirmation:= FALSE);
		END_IF
// 		bError 								:=	TRUE;
// 		udiErrorID							:=	322;
// 		sErrorDescription					:=	'Blokada wysunięcia szlabanu 2 - prawy - odblokuj';	
// 		sErrorDescription2					:=	'';			
	END_IF;
	// Alarm_0523	523	Error	Blokada schowania szlabanu 2 - prawy - odblokuj
	IF tonGate2OffError.Q THEN
		IF NOT arfbAlarm[3].bActive THEN
			arfbAlarm[3].Raise(nTimeStamp:=0);
		END_IF
	ELSE	
		IF  arfbAlarm[3].bActive AND bReset THEN
			arfbAlarm[3].Clear(nTimeStamp:=0, bResetConfirmation:= FALSE);
		END_IF
// 		bError 								:=	TRUE;
// 		udiErrorID							:=	323;
// 		sErrorDescription					:=	'Blokada schowania szlabanu 2 - prawy - odblokuj';	
// 		sErrorDescription2					:=	'';			
	END_IF;		
	// Alarm_0524	524	Error	Blokada wysunięcia tacki - odblokuj
	IF tonTrayOnError.Q THEN
		IF NOT arfbAlarm[4].bActive THEN
			arfbAlarm[4].Raise(nTimeStamp:=0);
		END_IF
	ELSE	
		IF  arfbAlarm[4].bActive AND bReset THEN
			arfbAlarm[4].Clear(nTimeStamp:=0, bResetConfirmation:= FALSE);
		END_IF
// 		bError 								:=	TRUE;
// 		udiErrorID							:=	324;
// 		sErrorDescription					:=	'Blokada wysunięcia tacki - odblokuj';	
// 		sErrorDescription2					:=	'';			
	END_IF;
	// Alarm_0525	525	Error	Blokada schowania tacki - odblokuj
	IF tonTrayOffError.Q THEN
		IF NOT arfbAlarm[5].bActive THEN
			arfbAlarm[5].Raise(nTimeStamp:=0);
		END_IF
	ELSE	
		IF  arfbAlarm[5].bActive AND bReset THEN
			arfbAlarm[5].Clear(nTimeStamp:=0, bResetConfirmation:= FALSE);
		END_IF
// 		bError 								:=	TRUE;
// 		udiErrorID							:=	325;
// 		sErrorDescription					:=	'Blokada schowania tacki - odblokuj';	
// 		sErrorDescription2					:=	'';			
	END_IF;		
	// Alarm_0526	526	Error	Blokada opuszczania wbijaka - odblokuj
	IF tonHammerOnError.Q THEN
		IF NOT arfbAlarm[6].bActive THEN
			arfbAlarm[6].Raise(nTimeStamp:=0);
		END_IF
	ELSE	
		IF  arfbAlarm[6].bActive AND bReset THEN
			arfbAlarm[6].Clear(nTimeStamp:=0, bResetConfirmation:= FALSE);
		END_IF
// 		bError 								:=	TRUE;
// 		udiErrorID							:=	326;
// 		sErrorDescription					:=	'Blokada opuszczania wbijaka - odblokuj';	
// 		sErrorDescription2					:=	'';			
	END_IF;
	// Alarm_0527	527	Error	Blokada podnoszenia wbijaka - odblokuj
	IF tonHammerOffError.Q THEN
		IF NOT arfbAlarm[7].bActive THEN
			arfbAlarm[7].Raise(nTimeStamp:=0);
		END_IF
	ELSE	
		IF  arfbAlarm[7].bActive AND bReset THEN
			arfbAlarm[7].Clear(nTimeStamp:=0, bResetConfirmation:= FALSE);
		END_IF
// 		bError 								:=	TRUE;
// 		udiErrorID							:=	327;
// 		sErrorDescription					:=	'Blokada podnoszenia wbijaka - odblokuj';	
// 		sErrorDescription2					:=	'';			
	END_IF;			
	// Alarm_0528	528	Error	Blokada wysunięcia pozycjonowania formatek - odblokuj
	IF tonFormPositioningOnError.Q THEN
		IF NOT arfbAlarm[8].bActive THEN
			arfbAlarm[8].Raise(nTimeStamp:=0);
		END_IF
	ELSE	
		IF  arfbAlarm[8].bActive AND bReset THEN
			arfbAlarm[8].Clear(nTimeStamp:=0, bResetConfirmation:= FALSE);
		END_IF
// 		bError 								:=	TRUE;
// 		udiErrorID							:=	328;
// 		sErrorDescription					:=	'Blokada wysunięcia pozycjonowania formatek - odblokuj';	
// 		sErrorDescription2					:=	'';			
	END_IF;
	// Alarm_0529	529	Error	Blokada schowania pozycjonowania formatek - odblokuj
	IF tonFormPositioningOffError.Q THEN
		IF NOT arfbAlarm[9].bActive THEN
			arfbAlarm[9].Raise(nTimeStamp:=0);
		END_IF
	ELSE	
		IF  arfbAlarm[9].bActive AND bReset THEN
			arfbAlarm[9].Clear(nTimeStamp:=0, bResetConfirmation:= FALSE);
		END_IF
// 		bError 								:=	TRUE;
// 		udiErrorID							:=	329;
// 		sErrorDescription					:=	'Blokada schowania pozycjonowania formatek - odblokuj';	
// 		sErrorDescription2					:=	'';			
	END_IF;		
	//Bląd braku opakowań w podajniku butelek
	// Alarm_0530	530	Error	Brak opakowań w podajniku - dołóż opakownia lub sprawdź ich ułożenie
	IF tonBottleAndFormTooLong.Q THEN
		IF NOT arfbAlarm[10].bActive THEN
			arfbAlarm[10].Raise(nTimeStamp:=0);
		END_IF
	ELSE	
		IF  arfbAlarm[10].bActive AND bReset THEN
			arfbAlarm[10].Clear(nTimeStamp:=0, bResetConfirmation:= FALSE);
		END_IF
// 		bError 								:=	TRUE;
// 		udiErrorID							:=	330;
// 		sErrorDescription					:=	'Brak opakowań w podajniku - dołóż opakownia lub sprawdź ich ułożenie';	
// 		sErrorDescription2					:=	'';			
	END_IF;	
	//Podnośnik nie porusza się pomimo wysterowania
	// Alarm_0531	531	Error	Blokada podnośnika lub brak zasilania - sprawdź czujnik lub odblokuj mechanicznie
	tonErrorHeightChange(IN:=(bHeightMotorUp OR bHeightMotorDown) AND nLastPositionHeightCV=lrHeightMotorCV, PT:=T#3S);
	IF tonErrorHeightChange.Q AND NOT bStateError THEN
		bHeightMotorUp						:=	FALSE;
		bHeightMotorDown					:=	FALSE;
		IF NOT arfbAlarm[11].bActive THEN
			arfbAlarm[11].Raise(nTimeStamp:=0);
		END_IF
	ELSE	
		IF  arfbAlarm[11].bActive AND bReset THEN
			arfbAlarm[11].Clear(nTimeStamp:=0, bResetConfirmation:= FALSE);
		END_IF
// 		bError								:=	TRUE;
// 		udiErrorID							:=	331;
// 		sErrorDescription					:=	'Blokada podnośnika lub brak zasilania - sprawdź czujnik lub odblokuj mechanicznie';	
	END_IF
	//Bład nastaw max
	// Alarm_0532	532	Error	Wartość zadana wysokości jest większa od maksymalnej - zmień ustawienia w recepturze {0}
	tonMaxHeight(IN:=lrHammerHeightSV>lrMaxHeight+1 AND bHomingDone AND lrMaxHeight>0 AND eState=E_Station.eReady,PT:=T#30S);
	IF tonMaxHeight.Q AND NOT bStateError THEN
		bHeightMotorUp						:=	FALSE;
		bHeightMotorDown					:=	FALSE;
		arfbAlarm[12].ipArguments.Clear() .AddInt(LREAL_TO_INT(lrMaxHeight));
		IF NOT arfbAlarm[12].bActive THEN
			arfbAlarm[12].Raise(nTimeStamp:=0);
		END_IF
	ELSE	
		IF  arfbAlarm[12].bActive AND bReset THEN
			arfbAlarm[12].Clear(nTimeStamp:=0, bResetConfirmation:= FALSE);
		END_IF
// 		bError								:=	TRUE;
// 		udiErrorID							:=	332;
// 		sErrorDescription					:=	'Wartość zadana wysokości jest większa od maksymalnej - zmień ustawienia w recepturze';
// 		sErrorDescription2					:=	REAL_TO_STRING(LREAL_TO_INT(lrMaxHeight));
	END_IF
	//Bład nastaw min
	// Alarm_0533	533	Error	Wartość zadana wysokości jest mniejsza od minimalnej - zmień ustawienia w recepturze {0}
	tonMinHeight(IN:=lrHammerHeightSV<lrMinHeight-1 AND bHomingDone AND lrMinHeight>0 AND eState=E_Station.eReady,PT:=T#30S);
	IF tonMinHeight.Q AND NOT bStateError THEN
		bHeightMotorUp						:=	FALSE;
		bHeightMotorDown					:=	FALSE;
		arfbAlarm[13].ipArguments.Clear() .AddInt(LREAL_TO_INT(lrMinHeight));
		IF NOT arfbAlarm[13].bActive THEN
			arfbAlarm[13].Raise(nTimeStamp:=0);
		END_IF
	ELSE	
		IF  arfbAlarm[13].bActive AND bReset THEN
			arfbAlarm[13].Clear(nTimeStamp:=0, bResetConfirmation:= FALSE);
		END_IF
// 		bError								:=	TRUE;
// 		udiErrorID							:=	333;
// 		sErrorDescription					:=	'Wartość zadana wysokości jest mniejsza od minimalnej - zmień ustawienia w recepturze';
// 		sErrorDescription2					:=	REAL_TO_STRING(LREAL_TO_INT(lrMinHeight));
	END_IF
	//Bład zbyt dużej różnicy nastaw
	// Alarm_0534	534	Error	Wartość aktualna jest zbyt różna od zadanej - zmień ustawienia w recepturze lub ustaw stację
	//tonSVCVDiffHeight(IN:=ABS(nPositionHeightSV-lrHeightMotorCV)>10 AND bHomingDone AND NOT bAlarmSVCVDiffHeightDisable AND eState=E_Station.eReady AND NOT bChangeOver2,PT:=T#5M);
	IF tonSVCVDiffHeight.Q AND NOT bStateError THEN
		bHeightMotorUp						:=	FALSE;
		bHeightMotorDown					:=	FALSE;
		arfbAlarm[14].ipArguments.Clear() .AddInt(LREAL_TO_INT(lrHammerHeightSV));
		IF NOT arfbAlarm[14].bActive THEN
			arfbAlarm[14].Raise(nTimeStamp:=0);
		END_IF
	ELSE	
		IF  arfbAlarm[14].bActive AND bReset THEN
			arfbAlarm[14].Clear(nTimeStamp:=0, bResetConfirmation:= FALSE);
		END_IF
// 		bError								:=	TRUE;
// 		udiErrorID							:=	334;
// 		sErrorDescription					:=	'Wartość aktualna jest zbyt różna od zadanej - zmień ustawienia w recepturze lub ustaw stację';
// 		sErrorDescription2					:=	REAL_TO_STRING(LREAL_TO_INT(lrHammerHeightSV));
	END_IF	
	//Błąd Serwa
	// Alarm_0535	535	Error	Błąd napędu karuzeli. Błąd NC: {0}
	tonWheelError(IN := stWheel.bError, PT:=T#2S);	
	IF tonWheelError.Q AND NOT bStateError (*AND NOT bWasEstop*) THEN
//		bHomingDone							:=	FALSE;
		//stWheel.mcReset.bExecute			:=	TRUE;
		arfbAlarm[15].ipArguments.Clear() .AddString(stWheel.stError.sNcError);
		IF NOT arfbAlarm[15].bActive THEN
			arfbAlarm[15].Raise(nTimeStamp:=0);
		END_IF
	ELSE	
		IF  arfbAlarm[15].bActive AND bReset THEN
			arfbAlarm[15].Clear(nTimeStamp:=0, bResetConfirmation:= FALSE);
		END_IF
// 		bError								:=	TRUE;
// 		udiErrorID							:=	335;
// 		sErrorDescription					:=	'Błąd napędu karuzeli. Błąd NC:';
// 		sErrorDescription2					:=	stWheel.stError.sNcError;
	END_IF
	//Błąd Falownika transportera
	// Alarm_0536	536	Error	Błąd falownika przenośnika butelek: {0} 
	IF fbConveyor.bError AND NOT bStateError AND NOT bWasEstop THEN
		fbConveyor.bRun						:= 	FALSE;
		arfbAlarm[16].ipArguments.Clear() .AddString(fbConveyor.sErrorDescription);
		IF NOT arfbAlarm[16].bActive THEN
			arfbAlarm[16].Raise(nTimeStamp:=0);
		END_IF
	ELSE	
		IF  arfbAlarm[16].bActive AND bReset THEN
			arfbAlarm[16].Clear(nTimeStamp:=0, bResetConfirmation:= FALSE);
		END_IF
// 		bError								:=	TRUE;
// 		udiErrorID							:=	336;
// 		sErrorDescription					:=	'Błąd falownika przenośnika butelek:';
// 		sErrorDescription2					:=	fbConveyor.sErrorDescription;
	END_IF
ELSE
	bError := FALSE;
END_IF

//-----------------------------------------------------------------------
IF bError AND NOT bStateError THEN

	IF eLastState = eRunning THEN
		bCycleNotDone						:= TRUE;
	END_IF

	eState 									:= E_Station.eError;
END_IF

//------------------------------------------------------------------------

(*Wyświetlanie błedu na wyjściu*)
bError;
FOR nAlarmNumerator := 0 TO 19 DO
	bError						:= bError OR arfbAlarm[nAlarmNumerator].bActive;
END_FOR
(*Przepisywanie nazwy stacji*)
sErrorStationName 							:= sStationName;

//Jezeli nie zbazowane to potrzebne bazowanie
IF NOT bHeightMotorEncoderHomed   THEN
	bHomingDone:=FALSE;
END_IF
END_ACTION

ACTION aHeightMotor:
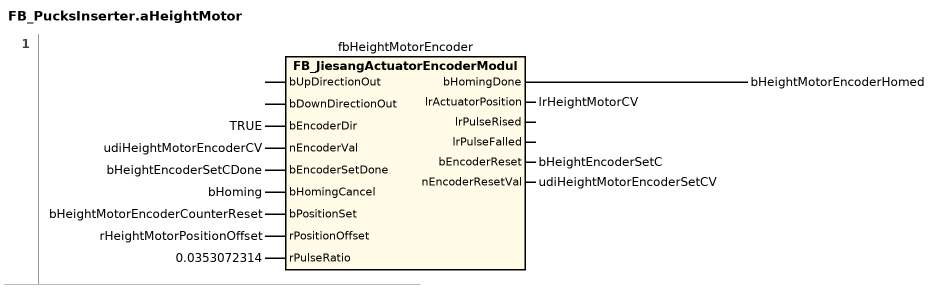
// NETWORK 1
fbHeightMotorEncoder(
    bEncoderDir := TRUE,
    nEncoderVal := udiHeightMotorEncoderCV,
    bEncoderSetDone := bHeightEncoderSetCDone,
    bHomingCancel := bHoming,
    bPositionSet := bHeightMotorEncoderCounterReset,
    rPositionOffset := rHeightMotorPositionOffset,
    rPulseRatio := 0.0353072314,
    lrActuatorPosition => lrHeightMotorCV,
    bEncoderReset => bHeightEncoderSetC,
    nEncoderResetVal => udiHeightMotorEncoderSetCV); // FB_JiesangActuatorEncoderModul
bHeightMotorEncoderHomed := fbHeightMotorEncoder.bHomingDone;
END_ACTION

ACTION aHoming:

stWheel.mcMoveRelative.lrAcceleration			:=	lrWheelAcceleration;
stWheel.mcMoveRelative.lrDeceleration			:=	lrWheelDeceleration;
stWheel.mcMoveRelative.lrJerk					:=	lrWheelJerk;
stWheel.mcMoveRelative.lrVelocity				:=	lrWheelVelocity;

stWheel.mcMoveVelocity.lrAcceleration			:= 	lrWheelAcceleration;
stWheel.mcMoveVelocity.lrDeceleration			:= 	lrWheelDeceleration;
stWheel.mcMoveVelocity.lrJerk					:= 	lrWheelJerk;
stWheel.mcMoveVelocity.lrVelocity				:= 	lrWheelVelocity;	

stWheel.stStatus.lrPosDiff;
stWheel.stStatus.lrActPos;

//Uwaga nie zmieniać czasu bo jednocześnie dwie stację jadą do góry
tofHeightMotorDown(IN:=bHeightMotorDown, PT:=T#1S); 
IF bHoming THEN 
	CASE iHomingStep OF
		0:
			bHomingDone										:=	FALSE;                                    		
			stWheel.mcMoveAbsolute.bExecute					:=	FALSE;
			stWheel.mcMoveRelative.bExecute					:=	FALSE;
			stWheel.mcMoveVelocity.bExecute					:=	FALSE;
			bHammer											:=	FALSE;
			IF bSensorHammerUp THEN
				iHomingStep									:=	iHomingStep	+	10;
			END_IF

		10:
			//IF NOT bSensorExitSensor OR NOT bSensorHoming THEN //Bazowanie pominete jak czujnik wyjsciowy zasłoniety
				bTray										:=	FALSE;
				IF bSensorTrayOff THEN
					iHomingStep								:=	iHomingStep +10;			
				END_IF
			//ELSE
			//	iHomingStep									:=	iHomingStep +10;			
			//END_IF

		20:
			//IF NOT bSensorExitSensor OR NOT bSensorHoming THEN //Bazowanie pominete jak czujnik wyjsciowy zasłoniety
				bGate1											:=	FALSE;
				bGate2											:=	FALSE;	
				IF bSensorGate1Off AND bSensorGate2Off THEN
					iHomingStep									:=	iHomingStep +10;		
				END_IF		
			//ELSE
			//	iHomingStep									:=	iHomingStep +10;			
			//END_IF
			
		30:
			bFormPositioning								:=	FALSE;
			IF bSensorFormPositioningOff THEN
				iHomingStep									:=	iHomingStep +10;		
			END_IF
			
		40:
//				fbHeightMotorEncoder.bHomingCancel		:= FALSE;
			//Podnoszenie stacji do maksymalnej pozycji
			IF NOT bHeightMotorEncoderHomed OR rtEncoderHomed.Q THEN
				bHeightMotorUp:= NOT tofHeightMotorDown.Q;;
				bHeightMotorDown:= FALSE;
				IF tonHeightNoChange.Q THEN
					bHeightMotorEncoderCounterReset:=TRUE;
					bHeightMotorUp:=FALSE;
				END_IF
				//Jesli enkoder zbazowany zakończ bazowanie	
				IF rtEncoderHomed.Q THEN
					bHeightMotorUp:=FALSE;
					bHeightMotorDown:=FALSE;
					//iHomingStep:=iHomingStep +10;
				END_IF		
					
			//Po podniesieniu stacji opuszczanie do ustalonej wysokości
			ELSIF bHeightMotorEncoderHomed THEN
				bHeightMotorEncoderCounterReset:=FALSE;
				bHeightMotorUp:=lrHeightMotorCV<=lrHammerHeightSV;
				bHeightMotorDown:=lrHeightMotorCV>=lrHammerHeightSV (*AND lrHeightMotorCV>=lrMinHeight*);
				//Kiedy stacja osiągnie wysokość zadaną
				IF ABS(lrHeightMotorCV-lrHammerHeightSV)<0.6 OR tonLimitPosMaxReachedDelay.Q OR tonLimitPosMinReachedDelay.Q (*OR lrHeightMotorCV>=lrMinHeight*) THEN
					bHeightMotorDown:=FALSE;
					bHeightMotorUp:=FALSE;
					iHomingStep:=iHomingStep +10;
				END_IF			
			END_IF
				
		50: //Sprawdzamy czy jest na czujniku

			IF bSensorHoming THEN
				iHomingStep									:= 60;
			ELSE                                        	
				iHomingStep									:= 70;
			END_IF
			
			//IF (bSensorExitSensor OR bSensorEntrySensor) AND bSensorHoming  THEN //Bazowanie pominete jak czujnik wyjsciowy zasłonietyTHEN	//Bazowanie pominete jak czujnik wyjsciowy zasłoniety
			//	iHomingStep									:= 110;
			//END_IF
			
		60: //Muszę wyjechać z czujnika
			stWheel.mcMoveRelative.lrAcceleration			:=	1500;
			stWheel.mcMoveRelative.lrDeceleration			:=	1500;
			stWheel.mcMoveRelative.lrJerk					:=	15000;
			stWheel.mcMoveRelative.lrVelocity				:=	15;
			stWheel.mcMoveRelative.lrDistance				:=	-15;
			stWheel.mcMoveRelative.bExecute					:= 	TRUE;

			
			IF stWheel.mcMoveRelative.bDone THEN
				stWheel.mcMoveRelative.bExecute				:= FALSE;
				iHomingStep									:= 70;
			END_IF
			
		70: //Bazuje na czujnik
			stWheel.mcMoveVelocity.lrAcceleration			:= 2500;
			stWheel.mcMoveVelocity.lrDeceleration			:= 2500;
			stWheel.mcMoveVelocity.lrJerk					:= 2500;
			stWheel.mcMoveVelocity.lrVelocity				:= 10;	
			stWheel.mcMoveVelocity.eDirection				:= MC_Positive_Direction; 
			stWheel.mcMoveVelocity.bExecute					:= TRUE;
			
			IF bSensorHoming THEN
				stWheel.mcMoveVelocity.bExecute				:= FALSE;
				iHomingStep									:= 80;
			END_IF
			
		80: //Zatrzymanie osi
			stWheel.mcStop.bExecute							:= TRUE;
			IF stWheel.mcStop.bDone THEN
				stWheel.mcStop.bExecute						:= FALSE;
				iHomingStep									:= 90;
			END_IF
	
		90:
			stWheel.mcHome.eHomingMode						:= MC_Direct;
			stWheel.mcHome.lrPosition						:= 0;
			stWheel.mcHome.bExecute							:= TRUE;
															
			IF stWheel.mcHome.bDone THEN             		
				stWheel.mcHome.bExecute						:= FALSE;
				iHomingStep									:= 100;
			END_IF
	
		100: 	
			stWheel.mcMoveAbsolute.lrAcceleration			:=1500;
			stWheel.mcMoveAbsolute.lrDeceleration			:=1500;
			stWheel.mcMoveAbsolute.lrJerk					:=15000;
			stWheel.mcMoveAbsolute.lrVelocity				:=15;
										  
			stWheel.mcMoveAbsolute.lrPosition			  	:= lrWheelOffset;
			stWheel.mcMoveAbsolute.bExecute				  	:= TRUE;
				
			IF stWheel.mcMoveAbsolute.bDone THEN
				lrWheelOffsetWhenHoming						:= lrWheelOffset;
				lrWheelLastKnownPosition					:= WheelAxisRef.NcToPlc.ModuloActPos;
				stWheel.mcMoveAbsolute.bExecute				:= FALSE;
				iHomingStep									:= 110;
			END_IF	
			
		110: //Bazujemy Enkoder
			stWheel.mcHome.eHomingMode						:= MC_Direct;
			stWheel.mcHome.lrPosition						:= 0;
			stWheel.mcHome.bExecute							:= TRUE;
															
			IF stWheel.mcHome.bDone THEN             		
				stWheel.mcHome.bExecute						:= FALSE;
				iHomingStep									:= 120;
			END_IF
			
		120:                             	
			iHomingStep										:= 130;
		
		130:
			iHomingStep										:= 140;
			
		140: //Zbazowano	
			iHomingStep										:=	0;
			eRunningState									:=	E_PuckInserterState.eReady;				
			eState											:=	E_Station.eHomingDone;
			
	END_CASE
END_IF
	
IF bHeightSet THEN

	//Podnoszenie stacji do maksymalnej pozycji
	IF NOT bHeightMotorEncoderHomed OR rtEncoderHomed.Q THEN
		bHeightMotorUp:= NOT tofHeightMotorDown.Q;;
		bHeightMotorDown:= FALSE;
		IF tonHeightNoChange.Q THEN
			bHeightMotorEncoderCounterReset:=TRUE;
			bHeightMotorUp:=FALSE;
		END_IF
		//Jesli enkoder zbazowany zakończ bazowanie	
		IF rtEncoderHomed.Q THEN
			bHeightMotorUp:=FALSE;
			bHeightMotorDown:=FALSE;
			eRunningState	:=	E_PuckInserterState.eReady;				
			eState			:=	E_Station.eHomingDone;
			iHomingStep:=0;
		END_IF		
			
	//Po podniesieniu stacji opuszczanie do ustalonej wysokości
	ELSIF bHeightMotorEncoderHomed THEN
		bHeightMotorEncoderCounterReset:=FALSE;
		bHeightMotorUp:=lrHeightMotorCV<=lrHammerHeightSV;
		bHeightMotorDown:=lrHeightMotorCV>=lrHammerHeightSV (*AND lrHeightMotorCV>=lrMinHeight*);
		//Kiedy stacja osiągnie wysokość zadaną
		IF ABS(lrHeightMotorCV-lrHammerHeightSV)<0.6 OR tonLimitPosMaxReachedDelay.Q OR tonLimitPosMinReachedDelay.Q (*OR lrHeightMotorCV>=lrMinHeight*) THEN
			bHeightMotorDown:=FALSE;
			bHeightMotorUp:=FALSE;
			eRunningState	:=	E_PuckInserterState.eReady;				
			eState			:=	E_Station.eHomingDone;
			iHomingStep:=0;	
		END_IF			
	END_IF
		
END_IF
END_ACTION

ACTION aInverter:
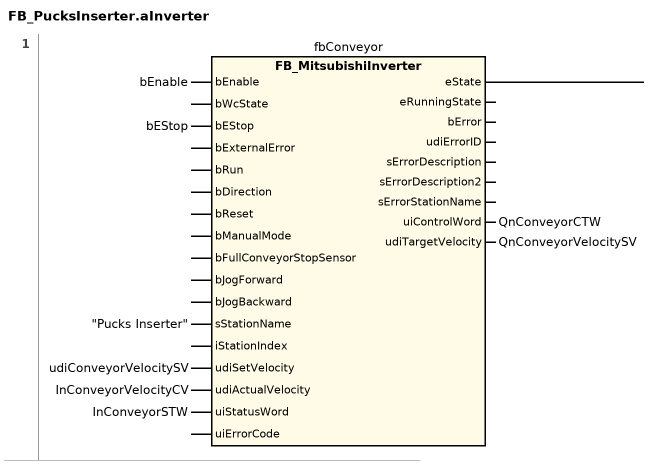
// NETWORK 1
fbConveyor(
    bEnable := bEnable,
    bEStop := bEStop,
    sStationName := "Pucks Inserter",
    udiSetVelocity := udiConveyorVelocitySV,
    udiActualVelocity := InConveyorVelocityCV,
    uiStatusWord := InConveyorSTW,
    uiControlWord => QnConveyorCTW,
    udiTargetVelocity => QnConveyorVelocitySV); // FB_MitsubishiInverter
END_ACTION

ACTION aLimits:
IF tAllowFormDelay<T#500MS THEN
	tAllowFormDelay:=T#500MS;
END_IF

IF tSensorFormDelay<T#50MS THEN
	tSensorFormDelay:=T#300MS;
END_IF

IF tSensorBottleDelay<T#0MS THEN
	tSensorBottleDelay:=T#0MS;
END_IF


IF udiConveyorVelocitySV < 100 	THEN udiConveyorVelocitySV := 100;	END_IF;
IF lrWheelAcceleration < 100 	THEN lrWheelAcceleration := 100;	END_IF;
IF lrWheelDeceleration < 100 	THEN lrWheelDeceleration := 100;	END_IF;
IF lrWheelJerk	< 100 			THEN lrWheelJerk := 100;			END_IF;
IF lrWheelVelocity	< 10 		THEN lrWheelVelocity := 10;			END_IF;
IF lrWheelOffset < -10			THEN lrWheelOffset	:= -10;			END_IF;
IF lrWheelOffset > 10			THEN lrWheelOffset	:= 10;			END_IF;


{warning 'dodać blokady w trybie manualnym żeby nie było kolicji'}
END_ACTION

ACTION aManualMovements:

IF NOT bRunPrepare AND NOT bRun AND bManualMovement THEN	
	stWheel.mcJog.bJogForward	:=	bManualWheelRight;
	stWheel.mcJog.bJogBackwards	:=	bManualWheelLeft;                                	                                  	                                   	
	bHammer						:=	bManualHammer;
	bHeightMotorUp				:=	bManualHeightMotorUp;
	bHeightMotorDown			:=	bManualHeightMotorDown;
	bTray						:=	bManuaTray;			
	bGate1						:=	bManualGate1;			
	bGate2						:=	bManualGate2;			
	bFormPositioning			:=	bManualFormPositioning;		
	fbConveyor.bRun				:=	bManualConveyor;				
ELSE
	bManualWheelRight			:=	FALSE;
	bManualWheelLeft			:=	FALSE;
	bManualHammer				:=	FALSE;
	bManualHeightMotorUp  		:=	FALSE;
	bManualHeightMotorDown		:=	FALSE;
	bManuaTray					:=	FALSE;
	bManualGate1				:=	FALSE;
	bManualGate2				:=	FALSE;
	bManualFormPositioning		:=	FALSE;
	bManualConveyor				:=	FALSE;	
END_IF

IF bHoming OR bHeightSet THEN
//	fbHeightMotorEncoder.bHomingCancel		:= TRUE;
	eState									:= E_Station.eHoming;
END_IF

IF NOT bEnable	THEN
	eState					:= E_Station.eReady;
END_IF
IF  (bRunPrepare OR bRun) AND bManualMovement THEN	
	aRunning();
END_IF
//IF bHeightMotorDown OR bHeightMotorUp THEN
//	bHomingDone					:=	FALSE;
//END_IF
//Zabezpieczenie przed kolizją stacji poprzez ruch podnośnika	
IF bHeightMotorDown AND lrHeightMotorCV<=lrMinHeight AND NOT bHoming AND NOT bHeightSet THEN
	bHeightMotorDown			:=	FALSE;
END_IF	

IF bHeightMotorUp AND lrHeightMotorCV>=lrMaxHeight AND NOT bHoming AND NOT bHeightSet THEN
	bHeightMotorUp				:=	FALSE;
END_IF	

IF NOT bRun THEN
	bCycleDone					:= FALSE;
	bCycleNotDone				:= FALSE;
END_IF
END_ACTION

ACTION aResetCommands:

stWheel.mcJog.bJogForward								:=	FALSE;
stWheel.mcJog.bJogBackwards								:=	FALSE;
stWheel.mcHome.bExecute									:=	FALSE;
                                                          	
stWheel.mcMoveAbsolute.bExecute							:=	FALSE;
stWheel.mcMoveRelative.bExecute							:=	FALSE;
stWheel.mcMoveVelocity.bExecute							:=	FALSE;
stWheel.mcMoveModulo.bExecute							:=	FALSE;
                                                          	
stWheel.mcHome.bExecute									:=	FALSE;
stWheel.mcStop.bExecute									:=	FALSE;
stWheel.mcReset.bExecute								:=	FALSE;
 
fbConveyor.bRun											:=	FALSE;

bHeightMotorUp											:=	FALSE;
bHeightMotorDown										:=	FALSE;

bHammer													:= FALSE;
bGate1													:= FALSE;
bGate2													:= FALSE;
bTray													:= FALSE;
bFormPositioning										:= FALSE;
                   
bManualHammer											:=	FALSE;
bManualHeightMotorUp									:=	FALSE;
bManualHeightMotorDown									:=	FALSE;
bManuaTray												:=	FALSE;
bManualGate1											:=	FALSE;
bManualGate2											:=	FALSE;
bManualFormPositioning									:=	FALSE;
bManualConveyor											:=	FALSE;
bManualWheelLeft 										:=	FALSE;
bManualWheelRight 										:=	FALSE;
//fbHeightMotorEncoder.bHomingCancel						:= FALSE;
				                          							  	
iHomingStep												:=	0;
                                                          	                            	
bResetCycleOn											:=	FALSE;	
iPreparingToMoveCase									:=	0;
iPreparingToReadyCase									:= 0;
END_ACTION

ACTION aResetCommandsNoTray:

stWheel.mcJog.bJogForward								:=	FALSE;
stWheel.mcJog.bJogBackwards								:=	FALSE;
stWheel.mcHome.bExecute									:=	FALSE;
                                                          	
stWheel.mcMoveAbsolute.bExecute							:=	FALSE;
stWheel.mcMoveRelative.bExecute							:=	FALSE;
stWheel.mcMoveVelocity.bExecute							:=	FALSE;
                                                          	
stWheel.mcHome.bExecute									:=	FALSE;
stWheel.mcStop.bExecute									:=	FALSE;
stWheel.mcReset.bExecute								:=	FALSE;
 
fbConveyor.bRun											:=	FALSE;

bHeightMotorUp											:=	FALSE;
bHeightMotorDown										:=	FALSE;

bHammer													:= FALSE;
bGate1													:= FALSE;
bGate2													:= FALSE;
//bTray													:= FALSE;
bFormPositioning										:= FALSE;
                   
bManualHammer											:=	FALSE;
bManualHeightMotorUp									:=	FALSE;
bManualHeightMotorDown									:=	FALSE;
bManuaTray												:=	FALSE;
bManualGate1											:=	FALSE;
bManualGate2											:=	FALSE;
bManualFormPositioning									:=	FALSE;
bManualConveyor											:=	FALSE;
bManualWheelLeft 										:=	FALSE;
bManualWheelRight 										:=	FALSE;
				                          							  	
iHomingStep												:=	0;
                                                          	                            	
bResetCycleOn											:=	FALSE;	
iPreparingToMoveCase									:=	0;
iPreparingToReadyCase									:= 0;
END_ACTION

ACTION aRunning:


CASE eRunningState OF

//--------------------------------------------------------------------------------------	
	//Pozycja gotowości 
	E_PuckInserterState.eReady:
	
		IF NOT bCycleDone AND NOT bCycleNotDone THEN	
			IF bRunPrepare OR bRun THEN
				eRunningState		:=	E_PuckInserterState.ePreparingToMove;
			END_IF
		END_IF
		bHammer						:=	FALSE;
		bGate1						:=	FALSE;
		bGate2						:=	FALSE;	
		bFormPositioning			:=	FALSE;			
//--------------------------------------------------------------------------------------	
	//Przygotowanie do ruchu
	E_PuckInserterState.ePreparingToMove:

		CASE iPreparingToMoveCase OF
			0:
				iPreparingToMoveCase := iPreparingToMoveCase + 10;
				
			10:
				IF bManualMode THEN
					iPreparingToMoveCase := iPreparingToMoveCase + 10;
				ELSE
					iPreparingToMoveCase := 100;
				END_IF
				
			20:
				(*
				IF  (
					(ABS(LMOD(WheelAxisRef.NcToPlc.ActPos,360.0/iWheelSlots)) > (360.0/iWheelSlots*0.01)) AND
					(ABS(LMOD(WheelAxisRef.NcToPlc.ActPos,360.0/iWheelSlots)) < (360.0/iWheelSlots*0.99))  
					)
					AND NOT (LMOD(WheelAxisRef.NcToPlc.ActPos,360.0/iWheelSlots) = 0) 
					THEN                       
						 stWheel.mcMoveAbsolute.lrPosition	:=	(WheelAxisRef.NcToPlc.ActPos+360.0/iWheelSlots-LMOD(WheelAxisRef.NcToPlc.ActPos,360.0/iWheelSlots))
							
						;
				ELSE
						stWheel.mcMoveAbsolute.lrPosition	:=	WheelAxisRef.NcToPlc.ActPos;				
				END_IF 
					stWheel.mcMoveAbsolute.bExecute			:=	TRUE;
					stWheel.mcMoveAbsolute.lrVelocity		:=	lrWheelVelocity / 2;
					stWheel.mcMoveAbsolute.lrAcceleration	:=	lrWheelAcceleration / 2;
					stWheel.mcMoveAbsolute.lrDeceleration	:=	lrWheelDeceleration / 2;
						
					IF stWheel.mcMoveAbsolute.bDone THEN	
						stWheel.mcMoveAbsolute.bExecute		:=	FALSE;
						iPreparingToMoveCase := 100;
					END_IF
				*)
				iPreparingToMoveCase := 100;
			100:
				//Transporter
				fbConveyor.bDirection 						:= FALSE;
				fbConveyor.bRun 							:= TRUE;
			
				//Decyzja
				IF tonBottleExitSensorDelay.Q AND bRun AND bEstopAndDoors THEN	// Jeżeli jest butelka to wbijaj
					iPreparingToMoveCase					:= 0;
					eRunningState							:= E_PuckInserterState.eGoAbove;
				ELSIF tonBottleEntrySensorDelay.Q AND (fbLevelSensor.bOut OR bManualMode) AND bRun AND bEstopAndDoors THEN	// Jeżeli nie ma butelki to obrót
					lrWheelLastKnownPosition				:= WheelAxisRef.NcToPlc.ModuloActPos;
					iPreparingToMoveCase					:= 0;					
					eRunningState							:= E_PuckInserterState.eTurning;
				END_IF
//				IF  tonFormsPresentDelay.Q  THEN
//					bFormPositioning						:=	TRUE;
//				END_IF				
				//Puść pusta formatkę
				IF tonAllowEmptyForm.Q THEN
					IF tonFormsPresentDelay.Q  THEN
						iPreparingToMoveCase				:= 0;						
						eRunningState						:= E_PuckInserterState.eBackToPosition;			
					END_IF
				END_IF	
			END_CASE
//--------------------------------------------------------------------------------------		
	E_PuckInserterState.eTurning:

		iTurningTest	:=	iTurningTest	+	1;

		bHammer						:=	 FALSE;
		bGate1						:=	 TRUE;
		bGate2						:=	 TRUE;
		bTray						:=	 TRUE;
		bFormPositioning			:=	 FALSE;

		//Karuzela
		stWheel.mcMoveRelative.lrAcceleration		:= lrWheelAcceleration;
		stWheel.mcMoveRelative.lrDeceleration		:= lrWheelDeceleration;
		stWheel.mcMoveRelative.lrJerk				:= lrWheelJerk;
		stWheel.mcMoveRelative.lrVelocity			:= lrWheelVelocity;
		
		
		
		IF 	lrWheelOffset<>lrWheelOffsetWhenHoming	THEN	
			bWheelOffsetChanged	:= TRUE;
		END_IF
		IF bWheelOffsetChanged THEN																														
			stWheel.mcMoveRelative.lrDistance		:= (360.0/INT_TO_LREAL(iWheelSlots)) + (lrWheelOffset-lrWheelOffsetWhenHoming);			
		ELSE
			stWheel.mcMoveRelative.lrDistance		:= (360.0/INT_TO_LREAL(iWheelSlots)) ;						
		END_IF
																	
		stWheel.mcMoveRelative.bExecute				:= TRUE;

			eRunningState							:=	E_PuckInserterState.eGoAbove;
 		
//--------------------------------------------------------------------------------------		
	E_PuckInserterState.eGoAbove:

		bHammer						:=	 FALSE;
		bGate1						:=	 TRUE;
		bGate2						:=	 TRUE;
		bTray						:=	 TRUE;
		bFormPositioning			:=	 FALSE;
		
		IF  tonFormsPresentDelay.Q  THEN
			eRunningState			:=	E_PuckInserterState.eCloseStoper;			
		END_IF
	

//-----------------------------------------------------------------------------------------
	E_PuckInserterState.eCloseStoper:		
	
		bFormPositioning							:=	TRUE;
		eRunningState								:=	E_PuckInserterState.eInsterting;
		

//------------------------------------------------------------------------------------	
	// Włóż butelek
	E_PuckInserterState.eInsterting:
	

		IF (stWheel.mcMoveRelative.bDone OR NOT stWheel.mcMoveRelative.bExecute) THEN
			bTray						:=	 FALSE;			
			stWheel.mcMoveRelative.bExecute			:=	FALSE;
			lrWheelOffsetWhenHoming					:=	lrWheelOffset;
			bWheelOffsetChanged						:=	FALSE;

		END_IF
		IF bSensorTrayOff AND NOT stWheel.mcMoveRelative.bExecute THEN
			bHammer					:= TRUE;			
		END_IF
		bGate1						:= TRUE;
		bGate2						:= TRUE;
		bTray						:= FALSE;
		//bFormPositioning			:= FALSE;		
		
		IF	((*ftIbSensorHammerDown.Q OR*) bSensorHammerDown)  THEN //Przeleciało przez czujnik albo jest	
			eRunningState			:=	E_PuckInserterState.eBackToPosition;	
		END_IF

//-----------------------------------------------------------------------------------	
	// Powrót do pozycji gotowości
	E_PuckInserterState.eBackToPosition:
	
		bHammer						:=	FALSE;
		bGate1						:=	FALSE;
		bGate2						:=	FALSE;	
		bFormPositioning			:=	FALSE;		
		
		IF bSensorHammerUp THEN
			lrWheelLastKnownPosition:= WheelAxisRef.NcToPlc.ModuloActPos;
			//bGate1					:=	TRUE;
			//bGate2					:=	TRUE;			
			//bTray					:= TRUE;
			bCycleDone				:=	TRUE;	
			eRunningState			:=	E_PuckInserterState.eReady;	
		END_IF
		
//-----------------------------------------------------------------------------------	

END_CASE
END_ACTION

ACTION aSignals:

	rtEncoderHomed				(CLK:=bHeightMotorEncoderHomed,Q=>);
	tonHeightNoChange			(IN:=((bHeightMotorUp OR bHeightMotorDown)	AND (nLastPositionHeightCV=lrHeightMotorCV)), PT:=T#1S); 
	tonLimitPosMinReachedDelay	(IN:=(lrHeightMotorCV<=lrMinHeight) 		AND eState=E_Station.eHoming,PT:=T#2S);
	tonLimitPosMaxReachedDelay	(IN:=(lrHeightMotorCV>=lrMaxHeight) 		AND eState=E_Station.eHoming,PT:=T#2S);
	tofMotorUpPermition			(IN:=bHeightMotorDown,									PT:=T#250MS);
	tofMotorDownPermition		(IN:=bHeightMotorUp,									PT:=T#250MS);	
	
	tonPreparingToDisabled		(IN:= eState = E_Station.ePreparingToDisable, 			PT:= T#1S);
	tonPreparingToReadyOn		(IN:= eState = E_Station.ePreparingToReady AND (iPreparingToReadyCase= 0 OR iPreparingToReadyCase= 15), 			PT:= T#2S);
	tofRunning					(IN:= eState = E_Station.eRunning, 						PT:= T#10S);	
	tonReady					(IN:= eState = E_Station.eReady, 						PT:= T#5S);	
	tonResetting				(IN:= eState = E_Station.eResetting,					PT:= T#200MS);
	rtResetCommands				(CLK:=eState = E_Station.eReady,						Q=>); 
	tonfbConveyorbRun 			(IN:=fbConveyor.bRun,									PT:=T#3S);                         	
	tonBottleEntrySensorDelay	(IN:= bSensorEntrySensor OR (bRun AND bManualMode) OR bSimulationSensor,	PT:=tSensorBottleDelay);
	tonBottleExitSensorDelay	(IN:= bSensorExitSensor (*OR (bRun AND bManualMode)*) (*OR bSimulationSensor*),		PT:=T#10MS);
	
	tonAllowEmptyForm 			(IN:= (NOT bSensorEntrySensor OR NOT  fbLevelSensor.bOut OR NOT bEstopAndDoors) AND bSensorFormPresent AND
								eRunningState = E_PuckInserterState.ePreparingToMove AND
								eState = E_Station.eRunning,
																			 		PT:=tAllowFormDelay);							
	
	tonFormsPresentDelay		(IN:= bSensorFormPresent OR (bRun AND bManualMode), 	PT:=tSensorFormDelay);

	ftIbSensorHammerDown		(CLK:= bSensorHammerDown,									Q=>);

	rtResetCycle				(CLK:= bResetCycle);

	tonArmDown					(IN:= bHammer, 										PT:=T#230MS);
	

	bSimulationSensor	:=	(bSimualtionMode OR bIgnoreError) AND NOT tonBottleEntrySensorDelay.Q;


	//Aktualna pozycja przeciągania
	lrWheelPositionCV	:=	stWheel.stStatus.lrActPos;
END_ACTION

ACTION aStationID:
udiStationID	:=	iStationIndex;
END_ACTION

ACTION aStatistic:

//Statystyka do zliczania czasu cyklu 
rtrigCycleTimerRead(CLK:=bCycleDone);

	IF rtrigCycleTimerRead.Q THEN
		tCycleTime:=tonCycleTimer.ET;
	END_IF
	
tonCycleTimer(IN:= eRunningState<>E_PuckInserterState.eReady AND eRunningState<>E_PuckInserterState.ePreparingToMove , PT:=T#1D);
END_ACTION

ACTION aStatus:

(*Zapisywanie ostatniego stanu*)
	IF eLastStateTemp<>eState THEN
		eLastState := eLastStateTemp;
	END_IF
	eLastStateTemp := eState;
	
	IF eLastRunningStateTemp<>eRunningState THEN
		eLastRunningState := eLastRunningStateTemp;
	END_IF
	eLastRunningStateTemp := eRunningState;
(*Koniec Zapisywanie ostatniego stanu*)
END_ACTION

ACTION aWarnings:

//Filtrowanie czujnika ultradźwiękowego

fbLevelSensor	(bIN:= (bSensorLevel OR bIgnoreError)(*AND tofRunning.Q*) AND tonfbConveyorbRun.Q, tFilterTimeOn:= T#3S, tFilterTimeOff:=T#400MS , bOUT=> );

IF NOT fbLevelSensor.bOUT THEN
	bWarning1						:=	TRUE;			
	udiWarningID					:=	1;
	sWarning1Description			:=	'Niski poziom butelek w sorterze butelek';
ELSE
	bWarning1						:=	FALSE;			
	udiWarningID					:=	0;
	sWarning1Description			:=	'';
END_IF

IF tofRunning.Q AND NOT bEstopAndDoors THEN
	bWarning2						:=	TRUE;	
	sWarning2Description			:=	'Otwarte drzwi';
ELSE
	bWarning2						:=	TRUE;	
	sWarning2Description			:=	'';
END_IF
END_ACTION

ACTION aWheelControlBlocks:
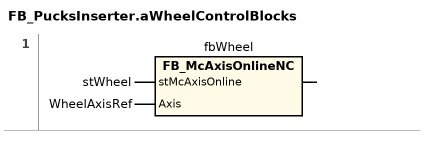
// NETWORK 1
fbWheel(stMcAxisOnline := stWheel, Axis := WheelAxisRef); // FB_McAxisOnlineNC
END_ACTION

ACTION fbwheel:
(*			IF mcWheelPower.Status THEN
				
				mcWheelMoveAbsolute.Execute:=TRUE;
			
